// Zapisywanie trybu pracy HC1 do pamięci urządzenia
IF xTrybPracyHC1Zapisz AND (fbTaktowanieZapisywaniaModbus.Q OR rtrigZapisModbus.Q) THEN
	fnModbusZapisRejestru(	bAdresUrzadzenia := bAdres,
							bFunkcja := INT_TO_BYTE(enumModbusKodyFunkcji.ZapisRejestru),
							uiAdresRejestru := uintTrybPracyHC1AdresModbus,
							pZmiennaReferencyjna := 0,
							wWartoscDoZapisania := REAL_TO_WORD(rTrybPracyHC1Zapis),
							intModbusOdczytZapisZadanieRozmiar := intModbusOdczytZapisZadanieRozmiar,
							arModbusOdczytZapisZadanie := arModbusOdczytZapisZadanie,
							intModbusOdczytZapisZadanieZnacznikZapisu := intModbusOdczytZapisZadanieZnacznikZapisu);
	IF intTrybPracyHC1 = REAL_TO_INT(rTrybPracyHC1Zapis) THEN					
		xTrybPracyHC1Zapisz := FALSE;
	END_IF
END_IF
// Temperatura punktu X2 krzywej grzewczej HC1
IF xKrzywaGrzewczaTemperaturyZewnetrznejX2HC1Zapisz AND (fbTaktowanieZapisywaniaModbus.Q OR rtrigZapisModbus.Q) THEN
	wKrzywaGrzewczaTemperaturyZewnetrznejX2HC1Zapis := fnOdwrocenieBitowTemperaturyUjemnejREAL_TO_WORD(rTemperaturaKelviny := rKrzywaGrzewczaTemperaturyZewnetrznejX2HC1Zapis);
	fnModbusZapisRejestru(	bAdresUrzadzenia := bAdres,
							bFunkcja := INT_TO_BYTE(enumModbusKodyFunkcji.ZapisRejestru),
							uiAdresRejestru := uintKrzywaGrzewczaTemperaturyZewnetrznejX2HC1AdresModbus,
							pZmiennaReferencyjna := 0,
							wWartoscDoZapisania := wKrzywaGrzewczaTemperaturyZewnetrznejX2HC1Zapis,
							intModbusOdczytZapisZadanieRozmiar := intModbusOdczytZapisZadanieRozmiar,
							arModbusOdczytZapisZadanie := arModbusOdczytZapisZadanie,
							intModbusOdczytZapisZadanieZnacznikZapisu := intModbusOdczytZapisZadanieZnacznikZapisu);
	IF rKrzywaGrzewczaTemperaturyZewnetrznejX2HC1 = rKrzywaGrzewczaTemperaturyZewnetrznejX2HC1Zapis THEN 						
		xKrzywaGrzewczaTemperaturyZewnetrznejX2HC1Zapisz := FALSE;
	END_IF
END_IF
// Temperatura punktu X3 krzywej grzewczej HC1
IF xKrzywaGrzewczaTemperaturyZewnetrznejX3HC1Zapisz AND (fbTaktowanieZapisywaniaModbus.Q OR rtrigZapisModbus.Q) THEN
	wKrzywaGrzewczaTemperaturyZewnetrznejX3HC1Zapis := fnOdwrocenieBitowTemperaturyUjemnejREAL_TO_WORD(rTemperaturaKelviny := rKrzywaGrzewczaTemperaturyZewnetrznejX3HC1Zapis);
	fnModbusZapisRejestru(	bAdresUrzadzenia := bAdres,
							bFunkcja := INT_TO_BYTE(enumModbusKodyFunkcji.ZapisRejestru),
							uiAdresRejestru := uintKrzywaGrzewczaTemperaturyZewnetrznejX3HC1AdresModbus,
							pZmiennaReferencyjna := 0,
							wWartoscDoZapisania := wKrzywaGrzewczaTemperaturyZewnetrznejX3HC1Zapis,
							intModbusOdczytZapisZadanieRozmiar := intModbusOdczytZapisZadanieRozmiar,
							arModbusOdczytZapisZadanie := arModbusOdczytZapisZadanie,
							intModbusOdczytZapisZadanieZnacznikZapisu := intModbusOdczytZapisZadanieZnacznikZapisu);
	IF rKrzywaGrzewczaTemperaturyZewnetrznejX3HC1 = rKrzywaGrzewczaTemperaturyZewnetrznejX3HC1Zapis THEN 						
		xKrzywaGrzewczaTemperaturyZewnetrznejX3HC1Zapisz := FALSE;
	END_IF
END_IF
// Temperatura punktu X4 krzywej grzewczej HC1
IF xKrzywaGrzewczaTemperaturyZewnetrznejX4HC1Zapisz AND (fbTaktowanieZapisywaniaModbus.Q OR rtrigZapisModbus.Q) THEN
	wKrzywaGrzewczaTemperaturyZewnetrznejX4HC1Zapis := fnOdwrocenieBitowTemperaturyUjemnejREAL_TO_WORD(rTemperaturaKelviny := rKrzywaGrzewczaTemperaturyZewnetrznejX4HC1Zapis);
	fnModbusZapisRejestru(	bAdresUrzadzenia := bAdres,
							bFunkcja := INT_TO_BYTE(enumModbusKodyFunkcji.ZapisRejestru),
							uiAdresRejestru := uintKrzywaGrzewczaTemperaturyZewnetrznejX4HC1AdresModbus,
							pZmiennaReferencyjna := 0,
							wWartoscDoZapisania := wKrzywaGrzewczaTemperaturyZewnetrznejX4HC1Zapis,
							intModbusOdczytZapisZadanieRozmiar := intModbusOdczytZapisZadanieRozmiar,
							arModbusOdczytZapisZadanie := arModbusOdczytZapisZadanie,
							intModbusOdczytZapisZadanieZnacznikZapisu := intModbusOdczytZapisZadanieZnacznikZapisu);
	IF rKrzywaGrzewczaTemperaturyZewnetrznejX4HC1 = rKrzywaGrzewczaTemperaturyZewnetrznejX4HC1Zapis THEN 						
		xKrzywaGrzewczaTemperaturyZewnetrznejX4HC1Zapisz := FALSE;
	END_IF
END_IF
// Temperatura punktu X5 krzywej grzewczej HC1
IF xKrzywaGrzewczaTemperaturyZewnetrznejX5HC1Zapisz AND (fbTaktowanieZapisywaniaModbus.Q OR rtrigZapisModbus.Q) THEN
	wKrzywaGrzewczaTemperaturyZewnetrznejX5HC1Zapis := fnOdwrocenieBitowTemperaturyUjemnejREAL_TO_WORD(rTemperaturaKelviny := rKrzywaGrzewczaTemperaturyZewnetrznejX5HC1Zapis);
	fnModbusZapisRejestru(	bAdresUrzadzenia := bAdres,
							bFunkcja := INT_TO_BYTE(enumModbusKodyFunkcji.ZapisRejestru),
							uiAdresRejestru := uintKrzywaGrzewczaTemperaturyZewnetrznejX5HC1AdresModbus,
							pZmiennaReferencyjna := 0,
							wWartoscDoZapisania := wKrzywaGrzewczaTemperaturyZewnetrznejX5HC1Zapis,
							intModbusOdczytZapisZadanieRozmiar := intModbusOdczytZapisZadanieRozmiar,
							arModbusOdczytZapisZadanie := arModbusOdczytZapisZadanie,
							intModbusOdczytZapisZadanieZnacznikZapisu := intModbusOdczytZapisZadanieZnacznikZapisu);
	IF rKrzywaGrzewczaTemperaturyZewnetrznejX5HC1 = rKrzywaGrzewczaTemperaturyZewnetrznejX5HC1Zapis THEN 						
		xKrzywaGrzewczaTemperaturyZewnetrznejX5HC1Zapisz := FALSE;
	END_IF
END_IF
// Temperatura punktu X6 krzywej grzewczej HC1
IF xKrzywaGrzewczaTemperaturyZewnetrznejX6HC1Zapisz AND (fbTaktowanieZapisywaniaModbus.Q OR rtrigZapisModbus.Q) THEN
	wKrzywaGrzewczaTemperaturyZewnetrznejX6HC1Zapis := fnOdwrocenieBitowTemperaturyUjemnejREAL_TO_WORD(rTemperaturaKelviny := rKrzywaGrzewczaTemperaturyZewnetrznejX6HC1Zapis);
	fnModbusZapisRejestru(	bAdresUrzadzenia := bAdres,
							bFunkcja := INT_TO_BYTE(enumModbusKodyFunkcji.ZapisRejestru),
							uiAdresRejestru := uintKrzywaGrzewczaTemperaturyZewnetrznejX6HC1AdresModbus,
							pZmiennaReferencyjna := 0,
							wWartoscDoZapisania := wKrzywaGrzewczaTemperaturyZewnetrznejX6HC1Zapis,
							intModbusOdczytZapisZadanieRozmiar := intModbusOdczytZapisZadanieRozmiar,
							arModbusOdczytZapisZadanie := arModbusOdczytZapisZadanie,
							intModbusOdczytZapisZadanieZnacznikZapisu := intModbusOdczytZapisZadanieZnacznikZapisu);
	IF rKrzywaGrzewczaTemperaturyZewnetrznejX6HC1 = rKrzywaGrzewczaTemperaturyZewnetrznejX6HC1Zapis THEN 						
		xKrzywaGrzewczaTemperaturyZewnetrznejX6HC1Zapisz := FALSE;
	END_IF
END_IF
// Temperatura punktu Y2 krzywej grzewczej HC1
IF xKrzywaGrzewczaTemperaturyZasilaniaY2HC1Zapisz AND (fbTaktowanieZapisywaniaModbus.Q OR rtrigZapisModbus.Q) THEN
	fnModbusZapisRejestru(	bAdresUrzadzenia := bAdres,
							bFunkcja := INT_TO_BYTE(enumModbusKodyFunkcji.ZapisRejestru),
							uiAdresRejestru := uintKrzywaGrzewczaTemperaturyZasilaniaY2HC1AdresModbus,
							pZmiennaReferencyjna := 0,
							wWartoscDoZapisania := REAL_TO_WORD((rKrzywaGrzewczaTemperaturyZasilaniaY2HC1Zapis - 273.15) * 10),
							intModbusOdczytZapisZadanieRozmiar := intModbusOdczytZapisZadanieRozmiar,
							arModbusOdczytZapisZadanie := arModbusOdczytZapisZadanie,
							intModbusOdczytZapisZadanieZnacznikZapisu := intModbusOdczytZapisZadanieZnacznikZapisu);
	IF rKrzywaGrzewczaTemperaturyZasilaniaY2HC1 = rKrzywaGrzewczaTemperaturyZasilaniaY2HC1Zapis THEN 						
		xKrzywaGrzewczaTemperaturyZasilaniaY2HC1Zapisz := FALSE;
	END_IF
END_IF
// Temperatura punktu Y3 krzywej grzewczej HC1
IF xKrzywaGrzewczaTemperaturyZasilaniaY3HC1Zapisz AND (fbTaktowanieZapisywaniaModbus.Q OR rtrigZapisModbus.Q) THEN
	fnModbusZapisRejestru(	bAdresUrzadzenia := bAdres,
							bFunkcja := INT_TO_BYTE(enumModbusKodyFunkcji.ZapisRejestru),
							uiAdresRejestru := uintKrzywaGrzewczaTemperaturyZasilaniaY3HC1AdresModbus,
							pZmiennaReferencyjna := 0,
							wWartoscDoZapisania := REAL_TO_WORD((rKrzywaGrzewczaTemperaturyZasilaniaY3HC1Zapis - 273.15) * 10),
							intModbusOdczytZapisZadanieRozmiar := intModbusOdczytZapisZadanieRozmiar,
							arModbusOdczytZapisZadanie := arModbusOdczytZapisZadanie,
							intModbusOdczytZapisZadanieZnacznikZapisu := intModbusOdczytZapisZadanieZnacznikZapisu);
	IF rKrzywaGrzewczaTemperaturyZasilaniaY3HC1 = rKrzywaGrzewczaTemperaturyZasilaniaY3HC1Zapis THEN 						
		xKrzywaGrzewczaTemperaturyZasilaniaY3HC1Zapisz := FALSE;
	END_IF
END_IF
// Temperatura punktu Y4 krzywej grzewczej HC1
IF xKrzywaGrzewczaTemperaturyZasilaniaY4HC1Zapisz AND (fbTaktowanieZapisywaniaModbus.Q OR rtrigZapisModbus.Q) THEN
	fnModbusZapisRejestru(	bAdresUrzadzenia := bAdres,
							bFunkcja := INT_TO_BYTE(enumModbusKodyFunkcji.ZapisRejestru),
							uiAdresRejestru := uintKrzywaGrzewczaTemperaturyZasilaniaY4HC1AdresModbus,
							pZmiennaReferencyjna := 0,
							wWartoscDoZapisania := REAL_TO_WORD((rKrzywaGrzewczaTemperaturyZasilaniaY4HC1Zapis - 273.15) * 10),
							intModbusOdczytZapisZadanieRozmiar := intModbusOdczytZapisZadanieRozmiar,
							arModbusOdczytZapisZadanie := arModbusOdczytZapisZadanie,
							intModbusOdczytZapisZadanieZnacznikZapisu := intModbusOdczytZapisZadanieZnacznikZapisu);
	IF rKrzywaGrzewczaTemperaturyZasilaniaY4HC1 = rKrzywaGrzewczaTemperaturyZasilaniaY4HC1Zapis THEN 						
		xKrzywaGrzewczaTemperaturyZasilaniaY4HC1Zapisz := FALSE;
	END_IF
END_IF
// Temperatura punktu Y5 krzywej grzewczej HC1
IF xKrzywaGrzewczaTemperaturyZasilaniaY5HC1Zapisz AND (fbTaktowanieZapisywaniaModbus.Q OR rtrigZapisModbus.Q) THEN
	fnModbusZapisRejestru(	bAdresUrzadzenia := bAdres,
							bFunkcja := INT_TO_BYTE(enumModbusKodyFunkcji.ZapisRejestru),
							uiAdresRejestru := uintKrzywaGrzewczaTemperaturyZasilaniaY5HC1AdresModbus,
							pZmiennaReferencyjna := 0,
							wWartoscDoZapisania := REAL_TO_WORD((rKrzywaGrzewczaTemperaturyZasilaniaY5HC1Zapis - 273.15) * 10),
							intModbusOdczytZapisZadanieRozmiar := intModbusOdczytZapisZadanieRozmiar,
							arModbusOdczytZapisZadanie := arModbusOdczytZapisZadanie,
							intModbusOdczytZapisZadanieZnacznikZapisu := intModbusOdczytZapisZadanieZnacznikZapisu);
	IF rKrzywaGrzewczaTemperaturyZasilaniaY5HC1 = rKrzywaGrzewczaTemperaturyZasilaniaY5HC1Zapis THEN 						
		xKrzywaGrzewczaTemperaturyZasilaniaY5HC1Zapisz := FALSE;
	END_IF
END_IF
// Temperatura punktu Y6 krzywej grzewczej HC1
IF xKrzywaGrzewczaTemperaturyZasilaniaY6HC1Zapisz AND (fbTaktowanieZapisywaniaModbus.Q OR rtrigZapisModbus.Q) THEN
	fnModbusZapisRejestru(	bAdresUrzadzenia := bAdres,
							bFunkcja := INT_TO_BYTE(enumModbusKodyFunkcji.ZapisRejestru),
							uiAdresRejestru := uintKrzywaGrzewczaTemperaturyZasilaniaY6HC1AdresModbus,
							pZmiennaReferencyjna := 0,
							wWartoscDoZapisania := REAL_TO_WORD((rKrzywaGrzewczaTemperaturyZasilaniaY6HC1Zapis - 273.15) * 10),
							intModbusOdczytZapisZadanieRozmiar := intModbusOdczytZapisZadanieRozmiar,
							arModbusOdczytZapisZadanie := arModbusOdczytZapisZadanie,
							intModbusOdczytZapisZadanieZnacznikZapisu := intModbusOdczytZapisZadanieZnacznikZapisu);
	IF rKrzywaGrzewczaTemperaturyZasilaniaY6HC1 = rKrzywaGrzewczaTemperaturyZasilaniaY6HC1Zapis THEN 						
		xKrzywaGrzewczaTemperaturyZasilaniaY6HC1Zapisz := FALSE;
	END_IF				
END_IF
// Zapisywanie trybu pracy DHW do pamięci urządzenia
IF xTrybPracyDHWZapisz AND (fbTaktowanieZapisywaniaModbus.Q OR rtrigZapisModbus.Q) THEN
	fnModbusZapisRejestru(	bAdresUrzadzenia := bAdres,
							bFunkcja := INT_TO_BYTE(enumModbusKodyFunkcji.ZapisRejestru),
							uiAdresRejestru := uintTrybPracyZadanieDHWAdresModbus,
							pZmiennaReferencyjna := 0,
							wWartoscDoZapisania := REAL_TO_WORD(rTrybPracyDHWZapis),
							intModbusOdczytZapisZadanieRozmiar := intModbusOdczytZapisZadanieRozmiar,
							arModbusOdczytZapisZadanie := arModbusOdczytZapisZadanie,
							intModbusOdczytZapisZadanieZnacznikZapisu := intModbusOdczytZapisZadanieZnacznikZapisu);
	IF intTrybPracyDHW = REAL_TO_INT(rTrybPracyDHWZapis) THEN					
		xTrybPracyDHWZapisz := FALSE;
	END_IF
END_IF

// Wyznaczanie okresu grzewczego
fbZegar15M(IN := NOT fbZegar15M.Q AND NOT xBladBrakZmianyTemperaturyZewnetrznej, PT := T#15M);

	// Obliczenie wschodu i zachodu słońca
fbWschodZachod(dtUTC_Time := WagoAppTime.FuGetDateAndTime(),
	rTimeZone := 0,
	xDST := FALSE,
	rLatitude := 54.441944,
	rLongitude := 18.559722);

	// Zapisywanie tempratury z 15-minutowym okresem, oraz obliczanie średniej
IF fbWschodZachod.dtUTC_Time > fbWschodZachod.dtSunrise AND fbWschodZachod.dtUTC_Time < fbWschodZachod.dtSunset THEN
	IF fbZegar15M.Q OR xPierwszySkan THEN
		aTemperatury[iTemperaturyIndex] := WORD_TO_REAL(wTemperaturaZewnetrzna) / 10;
		iTemperaturyIndex := iTemperaturyIndex + 1;
	END_IF	
	xObliczSrednia3Dni := TRUE;
ELSE 
	// Obliczanie średniej temperatury dziennej
	IF iTemperaturyIndex >= 40 THEN		// Oblicz średnią temperaturę tylko, jeśli zebranych zostało przynajmniej 40 próbek
		rTemperaturaSrednia1Dzien := 0;
		iIloscPomiarow := iTemperaturyIndex;
		FOR iTemperaturyIndex := 0 TO iIloscPomiarow BY 1 DO  
			rTemperaturaSrednia1Dzien := rTemperaturaSrednia1Dzien + aTemperatury[iTemperaturyIndex];
		END_FOR
		rTemperaturaSrednia1Dzien := rTemperaturaSrednia1Dzien / iTemperaturyIndex;
		xBladIloscPomiarowTemperatury := FALSE;
	ELSE
		rTemperaturaSrednia1Dzien := 15;
		xBladIloscPomiarowTemperatury := TRUE;
	END_IF
	// Obliczanie średniej z trzech dni
	IF xObliczSrednia3Dni THEN
		aTemperaturySrednie[iTemperaturySrednieIndex] := rTemperaturaSrednia1Dzien;
		iTemperaturySrednieIndex := iTemperaturySrednieIndex + 1;
		IF iTemperaturySrednieIndex = 3 THEN 
			iTemperaturySrednieIndex := 0;
			xTemperaturaSrednia3DniObliczona := TRUE;
		END_IF
		rTemperaturaSrednia3Dni := (aTemperaturySrednie[0] + aTemperaturySrednie[1] + aTemperaturySrednie[2]) / 3; 
		xObliczSrednia3Dni := FALSE;	
	END_IF
	iTemperaturyIndex := 0;
END_IF

	// Sprawdzenie warunku na włączenie ogrzewania (pomiędzy 15 września a 15 maja i/lub średnia temperatura jest poniżej 15 stopni)
IF  ((fbWschodZachod._rDay >= 15 AND fbWschodZachod._rMonth = 9) OR (fbWschodZachod._rMonth > 9 OR fbWschodZachod._rMonth < 5) OR (fbWschodZachod._rDay <= 15 AND fbWschodZachod._rMonth = 5)) OR 
	(rTemperaturaSrednia3Dni < 15 AND xTemperaturaSrednia3DniObliczona) OR xSezonGrzewczyCalyRok THEN
	xSezonGrzewczy := TRUE;
	intTrybPracyHC1Autonomizacja := enumPPPSWezelClimatixPOL63xTrybPracy.Komfort;
ELSE
	xSezonGrzewczy := FALSE;
	intTrybPracyHC1Autonomizacja := enumPPPSWezelClimatixPOL63xTrybPracy.OchronaBudynku;
END_IF

// dokonywanie obliczeń
(*
xOdczytanaKlasaAlarmuBezpieczenstwa := WORD_TO_BOOL(wOdczytanaKlasaAlarmuBezpieczenstwa);
xOdczytanaKlasaAlarmuKrytyczny := WORD_TO_BOOL(wOdczytanaKlasaAlarmuKrytyczny);
xOdczytanaKlasaAlarmuOstrzezenie := WORD_TO_BOOL(wOdczytanaKlasaAlarmuOstrzezenie);
xOdczytanaKlasaAlarmuInformacyjny := WORD_TO_BOOL(wOdczytanaKlasaAlarmuInformacyjny);
*)
xReczneWylaczenieInstalacji := WORD_TO_BOOL(wReczneWylaczenieInstalacji);

IF xInstalacjaHC1 OR xInstalacjaHC2 THEN
	fbTemperaturaZewnetrzna(	rWartoscWejsciowa := WORD_TO_REAL(wTemperaturaZewnetrzna),
									rDeadband := 0.5,
									tCzasMinimalny := tMinimalnyCzasRaportowania,
									tCzasMaksymalny := tMaksymalnyCzasRaportowania,
									rWynikMnoznik := 0.1,
									rWynikOffset := 273.15,
									rWartoscWejsciowaZaraportowana := rTemperaturaZewnetrznaZaraportowana,
									rWartoscWyjsciowa => rTemperaturaZewnetrzna);
END_IF

IF xInstalacjaHC1 THEN							
	fbTemperaturaGrzaniaNastawionaHC1(	rWartoscWejsciowa := WORD_TO_REAL(wTemperaturaGrzaniaNastawionaHC1),
									rDeadband := 0.5,
									tCzasMinimalny := tMinimalnyCzasRaportowania,
									tCzasMaksymalny := tMaksymalnyCzasRaportowania,
									rWynikMnoznik := 0.1,
									rWynikOffset := 273.15,
									rWartoscWejsciowaZaraportowana := rTemperaturaGrzaniaNastawionaHC1Zaraportowana,
									rWartoscWyjsciowa => rTemperaturaGrzaniaNastawionaHC1);
						
	fbTemperaturaGrzaniaNastawionaKrzywaGrzewczaHC1(	rWartoscWejsciowa := WORD_TO_REAL(wTemperaturaGrzaniaNastawionaKrzywaGrzewczaHC1),
									rDeadband := 0.5,
									tCzasMinimalny := tMinimalnyCzasRaportowania,
									tCzasMaksymalny := tMaksymalnyCzasRaportowania,
									rWynikMnoznik := 0.1,
									rWynikOffset := 273.15,
									rWartoscWejsciowaZaraportowana := rTemperaturaGrzaniaNastawionaKrzywaGrzewczaHC1Zaraportowana,
									rWartoscWyjsciowa => rTemperaturaGrzaniaNastawionaHC1);
	
	IF xReczneWylaczenieInstalacji THEN
		intTrybPracyHC1 := enumPPPSWezelClimatixPOL63xTrybPracy.ReczneWylaczenie;
	ELSE
		IF wTrybPracyHC1 = 0 THEN
			intTrybPracyHC1 := enumPPPSWezelClimatixPOL63xTrybPracy.Auto;
		ELSE
			IF wTrybPracyHC1 = 1 THEN
				intTrybPracyHC1 := enumPPPSWezelClimatixPOL63xTrybPracy.OchronaBudynku;
			ELSE
				IF wTrybPracyHC1 = 2 THEN
					intTrybPracyHC1 := enumPPPSWezelClimatixPOL63xTrybPracy.Ekonomiczny;
				ELSE
					IF wTrybPracyHC1 = 3 THEN
						intTrybPracyHC1 := enumPPPSWezelClimatixPOL63xTrybPracy.Komfort;
					END_IF
				END_IF
			END_IF
		END_IF
	END_IF
					
	fbTemperaturaGrzaniaNastawionaHC1(	rWartoscWejsciowa := WORD_TO_REAL(wTemperaturaGrzaniaNastawionaHC1),
									rDeadband := 0.5,
									tCzasMinimalny := tMinimalnyCzasRaportowania,
									tCzasMaksymalny := tMaksymalnyCzasRaportowania,
									rWynikMnoznik := 0.1,
									rWynikOffset := 273.15,
									rWartoscWejsciowaZaraportowana := rTemperaturaGrzaniaNastawionaHC1Zaraportowana,
									rWartoscWyjsciowa => rTemperaturaGrzaniaNastawionaHC1);

	fbTemperaturaGrzaniaNastawionaKrzywaGrzewczaHC1(	rWartoscWejsciowa := WORD_TO_REAL(wTemperaturaGrzaniaNastawionaKrzywaGrzewczaHC1),
									rDeadband := 0.5,
									tCzasMinimalny := tMinimalnyCzasRaportowania,
									tCzasMaksymalny := tMaksymalnyCzasRaportowania,
									rWynikMnoznik := 0.1,
									rWynikOffset := 273.15,
									rWartoscWejsciowaZaraportowana := rTemperaturaGrzaniaNastawionaKrzywaGrzewczaHC1Zaraportowana,
									rWartoscWyjsciowa => rTemperaturaGrzaniaNastawionaKrzywaGrzewczaHC1);
								
	fbTemperaturaZasilaniaObwoduHC1(	rWartoscWejsciowa := WORD_TO_REAL(wTemperaturaZasilaniaObwoduHC1),
									rDeadband := 0.5,
									tCzasMinimalny := tMinimalnyCzasRaportowania,
									tCzasMaksymalny := tMaksymalnyCzasRaportowania,
									rWynikMnoznik := 0.1,
									rWynikOffset := 273.15,
									rWartoscWejsciowaZaraportowana := rTemperaturaZasilaniaObwoduHC1Zaraportowana,
									rWartoscWyjsciowa => rTemperaturaZasilaniaObwoduHC1);
									
	fbTemperaturaPowrotuObwoduHC1(	rWartoscWejsciowa := WORD_TO_REAL(wTemperaturaPowrotuObwoduHC1),
									rDeadband := 0.5,
									tCzasMinimalny := tMinimalnyCzasRaportowania,
									tCzasMaksymalny := tMaksymalnyCzasRaportowania,
									rWynikMnoznik := 0.1,
									rWynikOffset := 273.15,
									rWartoscWejsciowaZaraportowana := rTemperaturaPowrotuObwoduHC1Zaraportowana,
									rWartoscWyjsciowa => rTemperaturaPowrotuObwoduHC1);
									
	fbTemperaturaPowrotuMiastoHC1(	rWartoscWejsciowa := WORD_TO_REAL(wTemperaturaPowrotuMiastoHC1),
									rDeadband := 0.5,
									tCzasMinimalny := tMinimalnyCzasRaportowania,
									tCzasMaksymalny := tMaksymalnyCzasRaportowania,
									rWynikMnoznik := 0.1,
									rWynikOffset := 273.15,
									rWartoscWejsciowaZaraportowana := rTemperaturaPowrotuMiastoHC1Zaraportowana,
									rWartoscWyjsciowa => rTemperaturaPowrotuMiastoHC1);
									
	fbTemperaturaZasilaniaBudynku(	rWartoscWejsciowa := WORD_TO_REAL(wTemperaturaZasilaniaBudynku),
									rDeadband := 0.5,
									tCzasMinimalny := tMinimalnyCzasRaportowania,
									tCzasMaksymalny := tMaksymalnyCzasRaportowania,
									rWynikMnoznik := 0.1,
									rWynikOffset := 273.15,
									rWartoscWejsciowaZaraportowana := rTemperaturaZasilaniaBudynkuZaraportowana,
									rWartoscWyjsciowa => rTemperaturaZasilaniaBudynku);
									
	fbTemperaturaPowrotuBudynku(	rWartoscWejsciowa := WORD_TO_REAL(wTemperaturaPowrotuBudynku),
									rDeadband := 0.5,
									tCzasMinimalny := tMinimalnyCzasRaportowania,
									tCzasMaksymalny := tMaksymalnyCzasRaportowania,
									rWynikMnoznik := 0.1,
									rWynikOffset := 273.15,
									rWartoscWejsciowaZaraportowana := rTemperaturaPowrotuBudynkuZaraportowana,
									rWartoscWyjsciowa => rTemperaturaPowrotuBudynku);
									
	fbSygnalZadaniaGrzaniaHC1(	rWartoscWejsciowa := WORD_TO_REAL(wSygnalZadaniaGrzaniaHC1),
									rDeadband := 0.05,
									tCzasMinimalny := tMinimalnyCzasRaportowania,
									tCzasMaksymalny := tMaksymalnyCzasRaportowania,
									rWynikMnoznik := 0.01,
									rWynikOffset := 0.0,
									rWartoscWejsciowaZaraportowana := rSygnalZadaniaGrzaniaHC1Zaraportowana,
									rWartoscWyjsciowa => rSygnalZadaniaGrzaniaHC1);
									
	fbStopienOtwarciaZaworuMiastoHC1(	rWartoscWejsciowa := WORD_TO_REAL(wStopienOtwarciaZaworuMiastoHC1),
									rDeadband := 0.05,
									tCzasMinimalny := tMinimalnyCzasRaportowania,
									tCzasMaksymalny := tMaksymalnyCzasRaportowania,
									rWynikMnoznik := 0.01,
									rWynikOffset := 0.0,
									rWartoscWejsciowaZaraportowana := rStopienOtwarciaZaworuMiastoHC1Zaraportowana,
									rWartoscWyjsciowa => rStopienOtwarciaZaworuMiastoHC1);
									
	IF wKrzywaGrzewczaTemperaturyZewnetrznejX2OdczytHC1 > 1000 THEN		// Jeśli temperatura ujemna odwróć bity	
		rKrzywaGrzewczaTemperaturyZewnetrznejX2HC1Raport := (-1) * WORD_TO_REAL(wKrzywaGrzewczaTemperaturyZewnetrznejX2OdczytHC1 XOR 16#FFFF);	
	ELSE
		rKrzywaGrzewczaTemperaturyZewnetrznejX2HC1Raport := WORD_TO_REAL(wKrzywaGrzewczaTemperaturyZewnetrznejX2OdczytHC1);
	END_IF		
	fbKrzywaGrzewczaTemperaturyZewnetrznejX2HC1(	rWartoscWejsciowa := rKrzywaGrzewczaTemperaturyZewnetrznejX2HC1Raport,
									rDeadband := 0.5,
									tCzasMinimalny := tMinimalnyCzasRaportowania,
									tCzasMaksymalny := tMaksymalnyCzasRaportowania,
									rWynikMnoznik := 0.1,
									rWynikOffset := 273.15,
									rWartoscWejsciowaZaraportowana := rKrzywaGrzewczaTemperaturyZewnetrznejX2HC1Zaraportowana,
									rWartoscWyjsciowa => rKrzywaGrzewczaTemperaturyZewnetrznejX2HC1);
	
	fbKrzywaGrzewczaTemperaturyZasilaniaY2HC1(	rWartoscWejsciowa := WORD_TO_REAL(wKrzywaGrzewczaTemperaturyZasilaniaY2OdczytHC1),
									rDeadband := 0.5,
									tCzasMinimalny := tMinimalnyCzasRaportowania,
									tCzasMaksymalny := tMaksymalnyCzasRaportowania,
									rWynikMnoznik := 0.1,
									rWynikOffset := 273.15,
									rWartoscWejsciowaZaraportowana := rKrzywaGrzewczaTemperaturyZasilaniaY2HC1Zaraportowana,
									rWartoscWyjsciowa => rKrzywaGrzewczaTemperaturyZasilaniaY2HC1);
	
	IF wKrzywaGrzewczaTemperaturyZewnetrznejX3OdczytHC1 > 1000 THEN		// Jeśli temperatura ujemna odwróć bity	
		rKrzywaGrzewczaTemperaturyZewnetrznejX3HC1Raport := (-1) * WORD_TO_REAL(wKrzywaGrzewczaTemperaturyZewnetrznejX3OdczytHC1 XOR 16#FFFF);	
	ELSE
		rKrzywaGrzewczaTemperaturyZewnetrznejX3HC1Raport := WORD_TO_REAL(wKrzywaGrzewczaTemperaturyZewnetrznejX3OdczytHC1);
	END_IF								
	fbKrzywaGrzewczaTemperaturyZewnetrznejX3HC1(	rWartoscWejsciowa := rKrzywaGrzewczaTemperaturyZewnetrznejX3HC1Raport,
									rDeadband := 0.5,
									tCzasMinimalny := tMinimalnyCzasRaportowania,
									tCzasMaksymalny := tMaksymalnyCzasRaportowania,
									rWynikMnoznik := 0.1,
									rWynikOffset := 273.15,
									rWartoscWejsciowaZaraportowana := rKrzywaGrzewczaTemperaturyZewnetrznejX3HC1Zaraportowana,
									rWartoscWyjsciowa => rKrzywaGrzewczaTemperaturyZewnetrznejX3HC1);
	
	fbKrzywaGrzewczaTemperaturyZasilaniaY3HC1(	rWartoscWejsciowa := WORD_TO_REAL(wKrzywaGrzewczaTemperaturyZasilaniaY3OdczytHC1),
									rDeadband := 0.5,
									tCzasMinimalny := tMinimalnyCzasRaportowania,
									tCzasMaksymalny := tMaksymalnyCzasRaportowania,
									rWynikMnoznik := 0.1,
									rWynikOffset := 273.15,
									rWartoscWejsciowaZaraportowana := rKrzywaGrzewczaTemperaturyZasilaniaY3HC1Zaraportowana,
									rWartoscWyjsciowa => rKrzywaGrzewczaTemperaturyZasilaniaY3HC1);
	
	IF wKrzywaGrzewczaTemperaturyZewnetrznejX4OdczytHC1 > 1000 THEN		// Jeśli temperatura ujemna odwróć bity	
		rKrzywaGrzewczaTemperaturyZewnetrznejX4HC1Raport := (-1) * WORD_TO_REAL(wKrzywaGrzewczaTemperaturyZewnetrznejX4OdczytHC1 XOR 16#FFFF);	
	ELSE
		rKrzywaGrzewczaTemperaturyZewnetrznejX4HC1Raport := WORD_TO_REAL(wKrzywaGrzewczaTemperaturyZewnetrznejX4OdczytHC1);
	END_IF												
	fbKrzywaGrzewczaTemperaturyZewnetrznejX4HC1(	rWartoscWejsciowa := rKrzywaGrzewczaTemperaturyZewnetrznejX4HC1Raport,
									rDeadband := 0.5,
									tCzasMinimalny := tMinimalnyCzasRaportowania,
									tCzasMaksymalny := tMaksymalnyCzasRaportowania,
									rWynikMnoznik := 0.1,
									rWynikOffset := 273.15,
									rWartoscWejsciowaZaraportowana := rKrzywaGrzewczaTemperaturyZewnetrznejX4HC1Zaraportowana,
									rWartoscWyjsciowa => rKrzywaGrzewczaTemperaturyZewnetrznejX4HC1);
	
	fbKrzywaGrzewczaTemperaturyZasilaniaY4HC1(	rWartoscWejsciowa := WORD_TO_REAL(wKrzywaGrzewczaTemperaturyZasilaniaY4OdczytHC1),
									rDeadband := 0.5,
									tCzasMinimalny := tMinimalnyCzasRaportowania,
									tCzasMaksymalny := tMaksymalnyCzasRaportowania,
									rWynikMnoznik := 0.1,
									rWynikOffset := 273.15,
									rWartoscWejsciowaZaraportowana := rKrzywaGrzewczaTemperaturyZasilaniaY4HC1Zaraportowana,
									rWartoscWyjsciowa => rKrzywaGrzewczaTemperaturyZasilaniaY4HC1);
	
		
	IF wKrzywaGrzewczaTemperaturyZewnetrznejX5OdczytHC1 > 1000 THEN		// Jeśli temperatura ujemna odwróć bity	
		rKrzywaGrzewczaTemperaturyZewnetrznejX5HC1Raport := (-1) * WORD_TO_REAL(wKrzywaGrzewczaTemperaturyZewnetrznejX5OdczytHC1 XOR 16#FFFF);	
	ELSE
		rKrzywaGrzewczaTemperaturyZewnetrznejX5HC1Raport := WORD_TO_REAL(wKrzywaGrzewczaTemperaturyZewnetrznejX5OdczytHC1);
	END_IF										
	fbKrzywaGrzewczaTemperaturyZewnetrznejX5HC1(	rWartoscWejsciowa := rKrzywaGrzewczaTemperaturyZewnetrznejX5HC1Raport,
									rDeadband := 0.5,
									tCzasMinimalny := tMinimalnyCzasRaportowania,
									tCzasMaksymalny := tMaksymalnyCzasRaportowania,
									rWynikMnoznik := 0.1,
									rWynikOffset := 273.15,
									rWartoscWejsciowaZaraportowana := rKrzywaGrzewczaTemperaturyZewnetrznejX5HC1Zaraportowana,
									rWartoscWyjsciowa => rKrzywaGrzewczaTemperaturyZewnetrznejX5HC1);
	
	fbKrzywaGrzewczaTemperaturyZasilaniaY5HC1(	rWartoscWejsciowa := WORD_TO_REAL(wKrzywaGrzewczaTemperaturyZasilaniaY5OdczytHC1),
									rDeadband := 0.5,
									tCzasMinimalny := tMinimalnyCzasRaportowania,
									tCzasMaksymalny := tMaksymalnyCzasRaportowania,
									rWynikMnoznik := 0.1,
									rWynikOffset := 273.15,
									rWartoscWejsciowaZaraportowana := rKrzywaGrzewczaTemperaturyZasilaniaY5HC1Zaraportowana,
									rWartoscWyjsciowa => rKrzywaGrzewczaTemperaturyZasilaniaY5HC1);
	
	IF wKrzywaGrzewczaTemperaturyZewnetrznejX6OdczytHC1 > 1000 THEN		// Jeśli temperatura ujemna odwróć bity	
		rKrzywaGrzewczaTemperaturyZewnetrznejX6HC1Raport := (-1) * WORD_TO_REAL(wKrzywaGrzewczaTemperaturyZewnetrznejX6OdczytHC1 XOR 16#FFFF);	
	ELSE
		rKrzywaGrzewczaTemperaturyZewnetrznejX6HC1Raport := WORD_TO_REAL(wKrzywaGrzewczaTemperaturyZewnetrznejX6OdczytHC1);
	END_IF									
	fbKrzywaGrzewczaTemperaturyZewnetrznejX6HC1(	rWartoscWejsciowa := rKrzywaGrzewczaTemperaturyZewnetrznejX6HC1Raport,
									rDeadband := 0.5,
									tCzasMinimalny := tMinimalnyCzasRaportowania,
									tCzasMaksymalny := tMaksymalnyCzasRaportowania,
									rWynikMnoznik := 0.1,
									rWynikOffset := 273.15,
									rWartoscWejsciowaZaraportowana := rKrzywaGrzewczaTemperaturyZewnetrznejX6HC1Zaraportowana,
									rWartoscWyjsciowa => rKrzywaGrzewczaTemperaturyZewnetrznejX6HC1);
	
	fbKrzywaGrzewczaTemperaturyZasilaniaY6HC1(	rWartoscWejsciowa := WORD_TO_REAL(wKrzywaGrzewczaTemperaturyZasilaniaY6OdczytHC1),
									rDeadband := 0.5,
									tCzasMinimalny := tMinimalnyCzasRaportowania,
									tCzasMaksymalny := tMaksymalnyCzasRaportowania,
									rWynikMnoznik := 0.1,
									rWynikOffset := 273.15,
									rWartoscWejsciowaZaraportowana := rKrzywaGrzewczaTemperaturyZasilaniaY6HC1Zaraportowana,
									rWartoscWyjsciowa => rKrzywaGrzewczaTemperaturyZasilaniaY6HC1);


	intTrybOperacjiHC1 := WORD_TO_INT(wTrybOperacjiHC1);
END_IF

IF xInstalacjaDHW THEN
	fbTemperaturaGrzaniaNastawionaDHW(	rWartoscWejsciowa := WORD_TO_REAL(wTemperaturaGrzaniaNastawionaDHW),
									rDeadband := 0.5,
									tCzasMinimalny := tMinimalnyCzasRaportowania,
									tCzasMaksymalny := tMaksymalnyCzasRaportowania,
									rWynikMnoznik := 0.1,
									rWynikOffset := 273.15,
									rWartoscWejsciowaZaraportowana := rTemperaturaGrzaniaNastawionaDHWZaraportowana,
									rWartoscWyjsciowa => rTemperaturaGrzaniaNastawionaDHW);
									
	IF xReczneWylaczenieInstalacji THEN
		intTrybPracyDHW := enumPPPSWezelClimatixPOL63xTrybPracy.ReczneWylaczenie;
	ELSE
		IF wTrybPracyDHW = 0 THEN
			intTrybPracyDHW := enumPPPSWezelClimatixPOL63xTrybPracy.Auto;
		ELSE
			IF wTrybPracyDHW = 1 THEN
				intTrybPracyDHW := enumPPPSWezelClimatixPOL63xTrybPracy.OchronaBudynku;
			ELSE
				IF wTrybPracyDHW = 2 THEN
					intTrybPracyDHW := enumPPPSWezelClimatixPOL63xTrybPracy.Ekonomiczny;
				ELSE
					IF wTrybPracyDHW = 3 THEN
						intTrybPracyDHW := enumPPPSWezelClimatixPOL63xTrybPracy.Komfort;
					END_IF
				END_IF
			END_IF
		END_IF
	END_IF
					
	fbTemperaturaPowrotuMiastoDHW(	rWartoscWejsciowa := WORD_TO_REAL(wTemperaturaPowrotuMiastoDHW),
									rDeadband := 0.5,
									tCzasMinimalny := tMinimalnyCzasRaportowania,
									tCzasMaksymalny := tMaksymalnyCzasRaportowania,
									rWynikMnoznik := 0.1,
									rWynikOffset := 273.15,
									rWartoscWejsciowaZaraportowana := rTemperaturaPowrotuMiastoDHWZaraportowana,
									rWartoscWyjsciowa => rTemperaturaPowrotuMiastoDHW);
									
	fbTemperaturaZasilaniaBudynekDHW(	rWartoscWejsciowa := WORD_TO_REAL(wTemperaturaZasilaniaBudynekDHW),
									rDeadband := 0.5,
									tCzasMinimalny := tMinimalnyCzasRaportowania,
									tCzasMaksymalny := tMaksymalnyCzasRaportowania,
									rWynikMnoznik := 0.1,
									rWynikOffset := 273.15,
									rWartoscWejsciowaZaraportowana := rTemperaturaZasilaniaBudynekDHWZaraportowana,
									rWartoscWyjsciowa => rTemperaturaZasilaniaBudynekDHW);
									
	fbTemperaturaPowrotuBudynekDHW(	rWartoscWejsciowa := WORD_TO_REAL(wTemperaturaPowrotuBudynekDHW),
									rDeadband := 0.5,
									tCzasMinimalny := tMinimalnyCzasRaportowania,
									tCzasMaksymalny := tMaksymalnyCzasRaportowania,
									rWynikMnoznik := 0.1,
									rWynikOffset := 273.15,
									rWartoscWejsciowaZaraportowana := rTemperaturaPowrotuBudynekDHWZaraportowana,
									rWartoscWyjsciowa => rTemperaturaPowrotuBudynekDHW);
									
	fbStopienOtwarciaZaworuMiastoDHW(	rWartoscWejsciowa := WORD_TO_REAL(wStopienOtwarciaZaworuMiastoDHW),
									rDeadband := 0.05,
									tCzasMinimalny := tMinimalnyCzasRaportowania,
									tCzasMaksymalny := tMaksymalnyCzasRaportowania,
									rWynikMnoznik := 0.01,
									rWynikOffset := 0.0,
									rWartoscWejsciowaZaraportowana := rStopienOtwarciaZaworuMiastoDHWZaraportowana,
									rWartoscWyjsciowa => rStopienOtwarciaZaworuMiastoDHW);
									
	intTrybOperacjiDHW := WORD_TO_INT(wTrybOperacjiDHW);
END_IF


//raportowanie
IF (intBlokadaWykonywaniaRozkazow <> intBlokadaWykonywaniaRozkazowZaraportowana OR rTemperaturaZewnetrzna <> rTemperaturaZewnetrznaZaraportowana OR rTemperaturaGrzaniaNastawionaHC1 <> rTemperaturaGrzaniaNastawionaHC1Zaraportowana
OR intTrybPracyHC1 <> intTrybPracyHC1Zaraportowana OR rTemperaturaZasilaniaObwoduHC1 <> rTemperaturaZasilaniaObwoduHC1Zaraportowana OR rTemperaturaPowrotuObwoduHC1 <> rTemperaturaPowrotuObwoduHC1Zaraportowana
OR rTemperaturaPowrotuMiastoHC1 <> rTemperaturaPowrotuMiastoHC1Zaraportowana OR rTemperaturaZasilaniaBudynku <> rTemperaturaZasilaniaBudynkuZaraportowana OR rTemperaturaPowrotuBudynku <> rTemperaturaPowrotuBudynkuZaraportowana
OR rSygnalZadaniaGrzaniaHC1 <> rSygnalZadaniaGrzaniaHC1Zaraportowana OR rStopienOtwarciaZaworuMiastoHC1 <> rStopienOtwarciaZaworuMiastoHC1Zaraportowana OR rKrzywaGrzewczaTemperaturyZewnetrznejX2HC1 <> rKrzywaGrzewczaTemperaturyZewnetrznejX2HC1Zaraportowana
OR rKrzywaGrzewczaTemperaturyZewnetrznejX2HC1 <> rKrzywaGrzewczaTemperaturyZewnetrznejX2HC1Zaraportowana OR rKrzywaGrzewczaTemperaturyZewnetrznejX3HC1 <> rKrzywaGrzewczaTemperaturyZewnetrznejX3HC1Zaraportowana OR rKrzywaGrzewczaTemperaturyZewnetrznejX4HC1 <> rKrzywaGrzewczaTemperaturyZewnetrznejX4HC1Zaraportowana
OR rKrzywaGrzewczaTemperaturyZewnetrznejX5HC1 <> rKrzywaGrzewczaTemperaturyZewnetrznejX5HC1Zaraportowana OR rKrzywaGrzewczaTemperaturyZewnetrznejX6HC1 <> rKrzywaGrzewczaTemperaturyZewnetrznejX6HC1Zaraportowana
OR rKrzywaGrzewczaTemperaturyZasilaniaY2HC1 <> rKrzywaGrzewczaTemperaturyZasilaniaY2HC1Zaraportowana OR rKrzywaGrzewczaTemperaturyZasilaniaY3HC1 <> rKrzywaGrzewczaTemperaturyZasilaniaY3HC1Zaraportowana OR rKrzywaGrzewczaTemperaturyZasilaniaY4HC1 <> rKrzywaGrzewczaTemperaturyZasilaniaY4HC1Zaraportowana
OR rKrzywaGrzewczaTemperaturyZasilaniaY5HC1 <> rKrzywaGrzewczaTemperaturyZasilaniaY5HC1Zaraportowana OR rKrzywaGrzewczaTemperaturyZasilaniaY6HC1 <> rKrzywaGrzewczaTemperaturyZasilaniaY6HC1Zaraportowana
OR rTemperaturaGrzaniaNastawionaDHW <> rTemperaturaGrzaniaNastawionaDHWZaraportowana OR intTrybPracyDHW <> intTrybPracyDHWZaraportowana OR rTemperaturaPowrotuMiastoDHW <> rTemperaturaPowrotuMiastoDHWZaraportowana
OR rTemperaturaZasilaniaBudynekDHW <> rTemperaturaZasilaniaBudynekDHWZaraportowana OR rTemperaturaPowrotuBudynekDHW <> rTemperaturaPowrotuBudynekDHWZaraportowana OR rStopienOtwarciaZaworuMiastoDHW <> rStopienOtwarciaZaworuMiastoDHWZaraportowana 
OR intTrybOperacjiHC1 <> intTrybOperacjiHC1Zaraportowana OR rTemperaturaGrzaniaNastawionaKrzywaGrzewczaHC1 <> rTemperaturaGrzaniaNastawionaKrzywaGrzewczaHC1Zaraportowana OR intTrybOperacjiDHW <> intTrybOperacjiDHWZaraportowana
OR intTrybOperacjiDHW <> intTrybOperacjiDHWZaraportowana OR wAlarmsWord1 <> wAlarmsWord1Zaraportowana OR wAlarmsWord2 <> wAlarmsWord2Zaraportowana OR wAlarmsWord3 <> wAlarmsWord3Zaraportowana
OR wAlarmsWord4 <> wAlarmsWord4Zaraportowana OR xSezonGrzewczy <> xSezonGrzewczyZaraportowana OR rTemperaturaSrednia1Dzien <> rTemperaturaSrednia1DzienZaraportowana) 
AND	arModbusStatusKomunikacji[bAdres] = enumModbusStatus.KomunikacjaPrawidlowa AND xPoInicjalizacji THEN
	xRaport := TRUE;
END_IF

IF xRaport THEN
	sDane := '';
	xRaport := FALSE;
	IF intBlokadaWykonywaniaRozkazow <> intBlokadaWykonywaniaRozkazowZaraportowana THEN
		intBlokadaWykonywaniaRozkazowZaraportowana := intBlokadaWykonywaniaRozkazow;
		fnKomunikatDaneDodaj_xOverFlow(sDane := sDane , sAtrybut := 'BLOK=' , sWartosc := INT_TO_STRING(intBlokadaWykonywaniaRozkazow) , xOverFlow := xOverFlow);	
			IF xOverFlow = TRUE THEN
				fnZapiszKomunikat(	sCalyKomunikat := '' ,
							sTypKomunikatu := 'A' ,
							sMnemonik := sMnemonik ,
							sMACAdres := sMACAdres ,
							sIDNadawcy := sIdInstancji ,
							sIDOdbiorcy := sIdAplikacji ,
							sDaneZapasowe := sDaneZapasowe ,
							sDane := sDane ,
							arTablicaKomunikatow := arTablicaKomunikatow ,
							intTablicaKomunikatowZnacznikZapisu := intTablicaKomunikatowZnacznikZapisu ,
							intTablicaKomunikatowRozmiar := intTablicaKomunikatowRozmiar ,
							sWyslanyKomunikat := sWyslanyKomunikatDummy);
				sDane := '';
			END_IF	
	END_IF	
	IF wAlarmsWord1 <> wAlarmsWord1Zaraportowana THEN
	wAlarmsWord1Zaraportowana := wAlarmsWord1;
	fnKomunikatDaneDodaj_xOverFlow(sDane := sDane , sAtrybut := 'ALARMWORD1=' , sWartosc := WORD_TO_STRING(wAlarmsWord1) , xOverFlow := xOverFlow);	
		IF xOverFlow = TRUE THEN
			fnZapiszKomunikat(	sCalyKomunikat := '' ,
						sTypKomunikatu := 'A' ,
						sMnemonik := sMnemonik ,
						sMACAdres := sMACAdres ,
						sIDNadawcy := sIdInstancji ,
						sIDOdbiorcy := sIdAplikacji ,
						sDaneZapasowe := sDaneZapasowe ,
						sDane := sDane ,
						arTablicaKomunikatow := arTablicaKomunikatow ,
						intTablicaKomunikatowZnacznikZapisu := intTablicaKomunikatowZnacznikZapisu ,
						intTablicaKomunikatowRozmiar := intTablicaKomunikatowRozmiar ,
						sWyslanyKomunikat := sWyslanyKomunikatDummy);
			sDane := '';
		END_IF	
	END_IF	
	IF wAlarmsWord2 <> wAlarmsWord2Zaraportowana THEN
	wAlarmsWord2Zaraportowana := wAlarmsWord2;
	fnKomunikatDaneDodaj_xOverFlow(sDane := sDane , sAtrybut := 'ALARMWORD2=' , sWartosc := WORD_TO_STRING(wAlarmsWord2) , xOverFlow := xOverFlow);	
		IF xOverFlow = TRUE THEN
			fnZapiszKomunikat(	sCalyKomunikat := '' ,
						sTypKomunikatu := 'A' ,
						sMnemonik := sMnemonik ,
						sMACAdres := sMACAdres ,
						sIDNadawcy := sIdInstancji ,
						sIDOdbiorcy := sIdAplikacji ,
						sDaneZapasowe := sDaneZapasowe ,
						sDane := sDane ,
						arTablicaKomunikatow := arTablicaKomunikatow ,
						intTablicaKomunikatowZnacznikZapisu := intTablicaKomunikatowZnacznikZapisu ,
						intTablicaKomunikatowRozmiar := intTablicaKomunikatowRozmiar ,
						sWyslanyKomunikat := sWyslanyKomunikatDummy);
			sDane := '';
		END_IF	
	END_IF	
	IF wAlarmsWord3 <> wAlarmsWord3Zaraportowana THEN
	wAlarmsWord3Zaraportowana := wAlarmsWord3;
	fnKomunikatDaneDodaj_xOverFlow(sDane := sDane , sAtrybut := 'ALARMWORD3=' , sWartosc := WORD_TO_STRING(wAlarmsWord3) , xOverFlow := xOverFlow);	
		IF xOverFlow = TRUE THEN
			fnZapiszKomunikat(	sCalyKomunikat := '' ,
						sTypKomunikatu := 'A' ,
						sMnemonik := sMnemonik ,
						sMACAdres := sMACAdres ,
						sIDNadawcy := sIdInstancji ,
						sIDOdbiorcy := sIdAplikacji ,
						sDaneZapasowe := sDaneZapasowe ,
						sDane := sDane ,
						arTablicaKomunikatow := arTablicaKomunikatow ,
						intTablicaKomunikatowZnacznikZapisu := intTablicaKomunikatowZnacznikZapisu ,
						intTablicaKomunikatowRozmiar := intTablicaKomunikatowRozmiar ,
						sWyslanyKomunikat := sWyslanyKomunikatDummy);
			sDane := '';
		END_IF	
	END_IF	
	IF wAlarmsWord4 <> wAlarmsWord4Zaraportowana THEN
	wAlarmsWord4Zaraportowana := wAlarmsWord4;
	fnKomunikatDaneDodaj_xOverFlow(sDane := sDane , sAtrybut := 'ALARMWORD4=' , sWartosc := WORD_TO_STRING(wAlarmsWord4) , xOverFlow := xOverFlow);	
		IF xOverFlow = TRUE THEN
			fnZapiszKomunikat(	sCalyKomunikat := '' ,
						sTypKomunikatu := 'A' ,
						sMnemonik := sMnemonik ,
						sMACAdres := sMACAdres ,
						sIDNadawcy := sIdInstancji ,
						sIDOdbiorcy := sIdAplikacji ,
						sDaneZapasowe := sDaneZapasowe ,
						sDane := sDane ,
						arTablicaKomunikatow := arTablicaKomunikatow ,
						intTablicaKomunikatowZnacznikZapisu := intTablicaKomunikatowZnacznikZapisu ,
						intTablicaKomunikatowRozmiar := intTablicaKomunikatowRozmiar ,
						sWyslanyKomunikat := sWyslanyKomunikatDummy);
			sDane := '';
		END_IF	
	END_IF	
	IF xInstalacjaHC1 OR xInstalacjaHC2 THEN
		IF rTemperaturaZewnetrzna <> rTemperaturaZewnetrznaZaraportowana AND arModbusStatusKomunikacji[bAdres] = enumModbusStatus.KomunikacjaPrawidlowa THEN
			rTemperaturaZewnetrznaZaraportowana := rTemperaturaZewnetrzna;
			fnKomunikatDaneDodaj_xOverFlow(sDane := sDane , sAtrybut := 'TEMPZEW=' , sWartosc := REAL_TO_STRING(rTemperaturaZewnetrzna) , xOverFlow := xOverFlow);	
			IF xOverFlow = TRUE THEN
				fnZapiszKomunikat(	sCalyKomunikat := '' ,
							sTypKomunikatu := 'A' ,
							sMnemonik := sMnemonik ,
							sMACAdres := sMACAdres ,
							sIDNadawcy := sIdInstancji ,
							sIDOdbiorcy := sIdAplikacji ,
							sDaneZapasowe := sDaneZapasowe ,
							sDane := sDane ,
							arTablicaKomunikatow := arTablicaKomunikatow ,
							intTablicaKomunikatowZnacznikZapisu := intTablicaKomunikatowZnacznikZapisu ,
							intTablicaKomunikatowRozmiar := intTablicaKomunikatowRozmiar ,
							sWyslanyKomunikat := sWyslanyKomunikatDummy);
				sDane := '';
			END_IF
		END_IF
	END_IF
	IF xInstalacjaHC1 THEN
		IF rTemperaturaGrzaniaNastawionaHC1 <> rTemperaturaGrzaniaNastawionaHC1Zaraportowana AND arModbusStatusKomunikacji[bAdres] = enumModbusStatus.KomunikacjaPrawidlowa THEN
			rTemperaturaGrzaniaNastawionaHC1Zaraportowana := rTemperaturaGrzaniaNastawionaHC1;
			fnKomunikatDaneDodaj_xOverFlow(sDane := sDane , sAtrybut := 'TEMPNASHC1=' , sWartosc := REAL_TO_STRING(rTemperaturaGrzaniaNastawionaHC1) , xOverFlow := xOverFlow);	
			IF xOverFlow = TRUE THEN
				fnZapiszKomunikat(	sCalyKomunikat := '' ,
							sTypKomunikatu := 'A' ,
							sMnemonik := sMnemonik ,
							sMACAdres := sMACAdres ,
							sIDNadawcy := sIdInstancji ,
							sIDOdbiorcy := sIdAplikacji ,
							sDaneZapasowe := sDaneZapasowe ,
							sDane := sDane ,
							arTablicaKomunikatow := arTablicaKomunikatow ,
							intTablicaKomunikatowZnacznikZapisu := intTablicaKomunikatowZnacznikZapisu ,
							intTablicaKomunikatowRozmiar := intTablicaKomunikatowRozmiar ,
							sWyslanyKomunikat := sWyslanyKomunikatDummy);
				sDane := '';
			END_IF
		END_IF
		IF rTemperaturaGrzaniaNastawionaKrzywaGrzewczaHC1 <> rTemperaturaGrzaniaNastawionaKrzywaGrzewczaHC1Zaraportowana AND arModbusStatusKomunikacji[bAdres] = enumModbusStatus.KomunikacjaPrawidlowa THEN
			rTemperaturaGrzaniaNastawionaKrzywaGrzewczaHC1Zaraportowana := rTemperaturaGrzaniaNastawionaKrzywaGrzewczaHC1;
			fnKomunikatDaneDodaj_xOverFlow(sDane := sDane , sAtrybut := 'TEMPNASKGHC1=' , sWartosc := REAL_TO_STRING(rTemperaturaGrzaniaNastawionaKrzywaGrzewczaHC1) , xOverFlow := xOverFlow);	
			IF xOverFlow = TRUE THEN
				fnZapiszKomunikat(	sCalyKomunikat := '' ,
							sTypKomunikatu := 'A' ,
							sMnemonik := sMnemonik ,
							sMACAdres := sMACAdres ,
							sIDNadawcy := sIdInstancji ,
							sIDOdbiorcy := sIdAplikacji ,
							sDaneZapasowe := sDaneZapasowe ,
							sDane := sDane ,
							arTablicaKomunikatow := arTablicaKomunikatow ,
							intTablicaKomunikatowZnacznikZapisu := intTablicaKomunikatowZnacznikZapisu ,
							intTablicaKomunikatowRozmiar := intTablicaKomunikatowRozmiar ,
							sWyslanyKomunikat := sWyslanyKomunikatDummy);
				sDane := '';
			END_IF
		END_IF
		IF intTrybPracyHC1 <> intTrybPracyHC1Zaraportowana AND arModbusStatusKomunikacji[bAdres] = enumModbusStatus.KomunikacjaPrawidlowa THEN
			intTrybPracyHC1Zaraportowana := intTrybPracyHC1;
			fnKomunikatDaneDodaj_xOverFlow(sDane := sDane , sAtrybut := 'TRYBNASHC1=' , sWartosc := INT_TO_STRING(intTrybPracyHC1) , xOverFlow := xOverFlow);	
			IF xOverFlow = TRUE THEN
				fnZapiszKomunikat(	sCalyKomunikat := '' ,
							sTypKomunikatu := 'A' ,
							sMnemonik := sMnemonik ,
							sMACAdres := sMACAdres ,
							sIDNadawcy := sIdInstancji ,
							sIDOdbiorcy := sIdAplikacji ,
							sDaneZapasowe := sDaneZapasowe ,
							sDane := sDane ,
							arTablicaKomunikatow := arTablicaKomunikatow ,
							intTablicaKomunikatowZnacznikZapisu := intTablicaKomunikatowZnacznikZapisu ,
							intTablicaKomunikatowRozmiar := intTablicaKomunikatowRozmiar ,
							sWyslanyKomunikat := sWyslanyKomunikatDummy);
				sDane := '';
			END_IF
		END_IF
		IF intTrybOperacjiHC1 <> intTrybOperacjiHC1Zaraportowana AND arModbusStatusKomunikacji[bAdres] = enumModbusStatus.KomunikacjaPrawidlowa THEN
			intTrybOperacjiHC1Zaraportowana := intTrybOperacjiHC1;
			fnKomunikatDaneDodaj_xOverFlow(sDane := sDane , sAtrybut := 'TRYBOPHC1=' , sWartosc := INT_TO_STRING(intTrybOperacjiHC1) , xOverFlow := xOverFlow);	
			IF xOverFlow = TRUE THEN
				fnZapiszKomunikat(	sCalyKomunikat := '' ,
							sTypKomunikatu := 'A' ,
							sMnemonik := sMnemonik ,
							sMACAdres := sMACAdres ,
							sIDNadawcy := sIdInstancji ,
							sIDOdbiorcy := sIdAplikacji ,
							sDaneZapasowe := sDaneZapasowe ,
							sDane := sDane ,
							arTablicaKomunikatow := arTablicaKomunikatow ,
							intTablicaKomunikatowZnacznikZapisu := intTablicaKomunikatowZnacznikZapisu ,
							intTablicaKomunikatowRozmiar := intTablicaKomunikatowRozmiar ,
							sWyslanyKomunikat := sWyslanyKomunikatDummy);
				sDane := '';
			END_IF
		END_IF
		IF rTemperaturaZasilaniaObwoduHC1 <> rTemperaturaZasilaniaObwoduHC1Zaraportowana AND arModbusStatusKomunikacji[bAdres] = enumModbusStatus.KomunikacjaPrawidlowa THEN
			rTemperaturaZasilaniaObwoduHC1Zaraportowana := rTemperaturaZasilaniaObwoduHC1;
			fnKomunikatDaneDodaj_xOverFlow(sDane := sDane , sAtrybut := 'TEMPZASOHC1=' , sWartosc := REAL_TO_STRING(rTemperaturaZasilaniaObwoduHC1) , xOverFlow := xOverFlow);	
			IF xOverFlow = TRUE THEN
				fnZapiszKomunikat(	sCalyKomunikat := '' ,
							sTypKomunikatu := 'A' ,
							sMnemonik := sMnemonik ,
							sMACAdres := sMACAdres ,
							sIDNadawcy := sIdInstancji ,
							sIDOdbiorcy := sIdAplikacji ,
							sDaneZapasowe := sDaneZapasowe ,
							sDane := sDane ,
							arTablicaKomunikatow := arTablicaKomunikatow ,
							intTablicaKomunikatowZnacznikZapisu := intTablicaKomunikatowZnacznikZapisu ,
							intTablicaKomunikatowRozmiar := intTablicaKomunikatowRozmiar ,
							sWyslanyKomunikat := sWyslanyKomunikatDummy);
				sDane := '';
			END_IF
		END_IF
		IF rTemperaturaPowrotuObwoduHC1 <> rTemperaturaPowrotuObwoduHC1Zaraportowana AND arModbusStatusKomunikacji[bAdres] = enumModbusStatus.KomunikacjaPrawidlowa THEN
			rTemperaturaPowrotuObwoduHC1Zaraportowana := rTemperaturaPowrotuObwoduHC1;
			fnKomunikatDaneDodaj_xOverFlow(sDane := sDane , sAtrybut := 'TEMPPOWOHC1=' , sWartosc := REAL_TO_STRING(rTemperaturaPowrotuObwoduHC1) , xOverFlow := xOverFlow);	
			IF xOverFlow = TRUE THEN
				fnZapiszKomunikat(	sCalyKomunikat := '' ,
							sTypKomunikatu := 'A' ,
							sMnemonik := sMnemonik ,
							sMACAdres := sMACAdres ,
							sIDNadawcy := sIdInstancji ,
							sIDOdbiorcy := sIdAplikacji ,
							sDaneZapasowe := sDaneZapasowe ,
							sDane := sDane ,
							arTablicaKomunikatow := arTablicaKomunikatow ,
							intTablicaKomunikatowZnacznikZapisu := intTablicaKomunikatowZnacznikZapisu ,
							intTablicaKomunikatowRozmiar := intTablicaKomunikatowRozmiar ,
							sWyslanyKomunikat := sWyslanyKomunikatDummy);
				sDane := '';
			END_IF
		END_IF
		IF rTemperaturaPowrotuMiastoHC1 <> rTemperaturaPowrotuMiastoHC1Zaraportowana AND arModbusStatusKomunikacji[bAdres] = enumModbusStatus.KomunikacjaPrawidlowa THEN
			rTemperaturaPowrotuMiastoHC1Zaraportowana := rTemperaturaPowrotuMiastoHC1;
			fnKomunikatDaneDodaj_xOverFlow(sDane := sDane , sAtrybut := 'TEMPPOWMHC1=' , sWartosc := REAL_TO_STRING(rTemperaturaPowrotuMiastoHC1) , xOverFlow := xOverFlow);	
			IF xOverFlow = TRUE THEN
				fnZapiszKomunikat(	sCalyKomunikat := '' ,
							sTypKomunikatu := 'A' ,
							sMnemonik := sMnemonik ,
							sMACAdres := sMACAdres ,
							sIDNadawcy := sIdInstancji ,
							sIDOdbiorcy := sIdAplikacji ,
							sDaneZapasowe := sDaneZapasowe ,
							sDane := sDane ,
							arTablicaKomunikatow := arTablicaKomunikatow ,
							intTablicaKomunikatowZnacznikZapisu := intTablicaKomunikatowZnacznikZapisu ,
							intTablicaKomunikatowRozmiar := intTablicaKomunikatowRozmiar ,
							sWyslanyKomunikat := sWyslanyKomunikatDummy);
				sDane := '';
			END_IF
		END_IF
		IF rTemperaturaZasilaniaBudynku <> rTemperaturaZasilaniaBudynkuZaraportowana AND arModbusStatusKomunikacji[bAdres] = enumModbusStatus.KomunikacjaPrawidlowa THEN
			rTemperaturaZasilaniaBudynkuZaraportowana := rTemperaturaZasilaniaBudynku;
			fnKomunikatDaneDodaj_xOverFlow(sDane := sDane , sAtrybut := 'TEMPZASB=' , sWartosc := REAL_TO_STRING(rTemperaturaZasilaniaBudynku) , xOverFlow := xOverFlow);	
			IF xOverFlow = TRUE THEN
				fnZapiszKomunikat(	sCalyKomunikat := '' ,
							sTypKomunikatu := 'A' ,
							sMnemonik := sMnemonik ,
							sMACAdres := sMACAdres ,
							sIDNadawcy := sIdInstancji ,
							sIDOdbiorcy := sIdAplikacji ,
							sDaneZapasowe := sDaneZapasowe ,
							sDane := sDane ,
							arTablicaKomunikatow := arTablicaKomunikatow ,
							intTablicaKomunikatowZnacznikZapisu := intTablicaKomunikatowZnacznikZapisu ,
							intTablicaKomunikatowRozmiar := intTablicaKomunikatowRozmiar ,
							sWyslanyKomunikat := sWyslanyKomunikatDummy);
				sDane := '';
			END_IF
		END_IF
		IF rTemperaturaPowrotuBudynku <> rTemperaturaPowrotuBudynkuZaraportowana AND arModbusStatusKomunikacji[bAdres] = enumModbusStatus.KomunikacjaPrawidlowa THEN
			rTemperaturaPowrotuBudynkuZaraportowana := rTemperaturaPowrotuBudynku;
			fnKomunikatDaneDodaj_xOverFlow(sDane := sDane , sAtrybut := 'TEMPPOWB=' , sWartosc := REAL_TO_STRING(rTemperaturaPowrotuBudynku) , xOverFlow := xOverFlow);	
			IF xOverFlow = TRUE THEN
				fnZapiszKomunikat(	sCalyKomunikat := '' ,
							sTypKomunikatu := 'A' ,
							sMnemonik := sMnemonik ,
							sMACAdres := sMACAdres ,
							sIDNadawcy := sIdInstancji ,
							sIDOdbiorcy := sIdAplikacji ,
							sDaneZapasowe := sDaneZapasowe ,
							sDane := sDane ,
							arTablicaKomunikatow := arTablicaKomunikatow ,
							intTablicaKomunikatowZnacznikZapisu := intTablicaKomunikatowZnacznikZapisu ,
							intTablicaKomunikatowRozmiar := intTablicaKomunikatowRozmiar ,
							sWyslanyKomunikat := sWyslanyKomunikatDummy);
				sDane := '';
			END_IF
		END_IF
		IF rSygnalZadaniaGrzaniaHC1 <> rSygnalZadaniaGrzaniaHC1Zaraportowana AND arModbusStatusKomunikacji[bAdres] = enumModbusStatus.KomunikacjaPrawidlowa THEN
			rSygnalZadaniaGrzaniaHC1Zaraportowana := rSygnalZadaniaGrzaniaHC1;
			fnKomunikatDaneDodaj_xOverFlow(sDane := sDane , sAtrybut := 'STERGRZHC1=' , sWartosc := REAL_TO_STRING(rSygnalZadaniaGrzaniaHC1) , xOverFlow := xOverFlow);	
			IF xOverFlow = TRUE THEN
				fnZapiszKomunikat(	sCalyKomunikat := '' ,
							sTypKomunikatu := 'A' ,
							sMnemonik := sMnemonik ,
							sMACAdres := sMACAdres ,
							sIDNadawcy := sIdInstancji ,
							sIDOdbiorcy := sIdAplikacji ,
							sDaneZapasowe := sDaneZapasowe ,
							sDane := sDane ,
							arTablicaKomunikatow := arTablicaKomunikatow ,
							intTablicaKomunikatowZnacznikZapisu := intTablicaKomunikatowZnacznikZapisu ,
							intTablicaKomunikatowRozmiar := intTablicaKomunikatowRozmiar ,
							sWyslanyKomunikat := sWyslanyKomunikatDummy);
				sDane := '';
			END_IF
		END_IF
		IF rStopienOtwarciaZaworuMiastoHC1 <> rStopienOtwarciaZaworuMiastoHC1Zaraportowana AND arModbusStatusKomunikacji[bAdres] = enumModbusStatus.KomunikacjaPrawidlowa THEN
			rStopienOtwarciaZaworuMiastoHC1Zaraportowana := rStopienOtwarciaZaworuMiastoHC1;
			fnKomunikatDaneDodaj_xOverFlow(sDane := sDane , sAtrybut := 'STERZAWMHC1=' , sWartosc := REAL_TO_STRING(rStopienOtwarciaZaworuMiastoHC1) , xOverFlow := xOverFlow);	
			IF xOverFlow = TRUE THEN
				fnZapiszKomunikat(	sCalyKomunikat := '' ,
							sTypKomunikatu := 'A' ,
							sMnemonik := sMnemonik ,
							sMACAdres := sMACAdres ,
							sIDNadawcy := sIdInstancji ,
							sIDOdbiorcy := sIdAplikacji ,
							sDaneZapasowe := sDaneZapasowe ,
							sDane := sDane ,
							arTablicaKomunikatow := arTablicaKomunikatow ,
							intTablicaKomunikatowZnacznikZapisu := intTablicaKomunikatowZnacznikZapisu ,
							intTablicaKomunikatowRozmiar := intTablicaKomunikatowRozmiar ,
							sWyslanyKomunikat := sWyslanyKomunikatDummy);
				sDane := '';
			END_IF
		END_IF
		IF rKrzywaGrzewczaTemperaturyZewnetrznejX2HC1 <> rKrzywaGrzewczaTemperaturyZewnetrznejX2HC1Zaraportowana AND arModbusStatusKomunikacji[bAdres] = enumModbusStatus.KomunikacjaPrawidlowa THEN
			rKrzywaGrzewczaTemperaturyZewnetrznejX2HC1Zaraportowana := rKrzywaGrzewczaTemperaturyZewnetrznejX2HC1;
			fnKomunikatDaneDodaj_xOverFlow(sDane := sDane , sAtrybut := 'TEMPKGHC1X2=' , sWartosc := REAL_TO_STRING(rKrzywaGrzewczaTemperaturyZewnetrznejX2HC1) , xOverFlow := xOverFlow);	
			IF xOverFlow = TRUE THEN
				fnZapiszKomunikat(	sCalyKomunikat := '' ,
							sTypKomunikatu := 'A' ,
							sMnemonik := sMnemonik ,
							sMACAdres := sMACAdres ,
							sIDNadawcy := sIdInstancji ,
							sIDOdbiorcy := sIdAplikacji ,
							sDaneZapasowe := sDaneZapasowe ,
							sDane := sDane ,
							arTablicaKomunikatow := arTablicaKomunikatow ,
							intTablicaKomunikatowZnacznikZapisu := intTablicaKomunikatowZnacznikZapisu ,
							intTablicaKomunikatowRozmiar := intTablicaKomunikatowRozmiar ,
							sWyslanyKomunikat := sWyslanyKomunikatDummy);
				sDane := '';
			END_IF
		END_IF
		IF rKrzywaGrzewczaTemperaturyZewnetrznejX3HC1 <> rKrzywaGrzewczaTemperaturyZewnetrznejX3HC1Zaraportowana AND arModbusStatusKomunikacji[bAdres] = enumModbusStatus.KomunikacjaPrawidlowa THEN
			rKrzywaGrzewczaTemperaturyZewnetrznejX3HC1Zaraportowana := rKrzywaGrzewczaTemperaturyZewnetrznejX3HC1;
			fnKomunikatDaneDodaj_xOverFlow(sDane := sDane , sAtrybut := 'TEMPKGHC1X3=' , sWartosc := REAL_TO_STRING(rKrzywaGrzewczaTemperaturyZewnetrznejX3HC1) , xOverFlow := xOverFlow);	
			IF xOverFlow = TRUE THEN
				fnZapiszKomunikat(	sCalyKomunikat := '' ,
							sTypKomunikatu := 'A' ,
							sMnemonik := sMnemonik ,
							sMACAdres := sMACAdres ,
							sIDNadawcy := sIdInstancji ,
							sIDOdbiorcy := sIdAplikacji ,
							sDaneZapasowe := sDaneZapasowe ,
							sDane := sDane ,
							arTablicaKomunikatow := arTablicaKomunikatow ,
							intTablicaKomunikatowZnacznikZapisu := intTablicaKomunikatowZnacznikZapisu ,
							intTablicaKomunikatowRozmiar := intTablicaKomunikatowRozmiar ,
							sWyslanyKomunikat := sWyslanyKomunikatDummy);
				sDane := '';
			END_IF
		END_IF
		IF rKrzywaGrzewczaTemperaturyZewnetrznejX4HC1 <> rKrzywaGrzewczaTemperaturyZewnetrznejX4HC1Zaraportowana AND arModbusStatusKomunikacji[bAdres] = enumModbusStatus.KomunikacjaPrawidlowa THEN
			rKrzywaGrzewczaTemperaturyZewnetrznejX4HC1Zaraportowana := rKrzywaGrzewczaTemperaturyZewnetrznejX4HC1;
			fnKomunikatDaneDodaj_xOverFlow(sDane := sDane , sAtrybut := 'TEMPKGHC1X4=' , sWartosc := REAL_TO_STRING(rKrzywaGrzewczaTemperaturyZewnetrznejX4HC1) , xOverFlow := xOverFlow);	
			IF xOverFlow = TRUE THEN
				fnZapiszKomunikat(	sCalyKomunikat := '' ,
							sTypKomunikatu := 'A' ,
							sMnemonik := sMnemonik ,
							sMACAdres := sMACAdres ,
							sIDNadawcy := sIdInstancji ,
							sIDOdbiorcy := sIdAplikacji ,
							sDaneZapasowe := sDaneZapasowe ,
							sDane := sDane ,
							arTablicaKomunikatow := arTablicaKomunikatow ,
							intTablicaKomunikatowZnacznikZapisu := intTablicaKomunikatowZnacznikZapisu ,
							intTablicaKomunikatowRozmiar := intTablicaKomunikatowRozmiar ,
							sWyslanyKomunikat := sWyslanyKomunikatDummy);
				sDane := '';
			END_IF
		END_IF
		IF rKrzywaGrzewczaTemperaturyZewnetrznejX5HC1 <> rKrzywaGrzewczaTemperaturyZewnetrznejX5HC1Zaraportowana AND arModbusStatusKomunikacji[bAdres] = enumModbusStatus.KomunikacjaPrawidlowa THEN
			rKrzywaGrzewczaTemperaturyZewnetrznejX5HC1Zaraportowana := rKrzywaGrzewczaTemperaturyZewnetrznejX5HC1;
			fnKomunikatDaneDodaj_xOverFlow(sDane := sDane , sAtrybut := 'TEMPKGHC1X5=' , sWartosc := REAL_TO_STRING(rKrzywaGrzewczaTemperaturyZewnetrznejX5HC1) , xOverFlow := xOverFlow);	
			IF xOverFlow = TRUE THEN
				fnZapiszKomunikat(	sCalyKomunikat := '' ,
							sTypKomunikatu := 'A' ,
							sMnemonik := sMnemonik ,
							sMACAdres := sMACAdres ,
							sIDNadawcy := sIdInstancji ,
							sIDOdbiorcy := sIdAplikacji ,
							sDaneZapasowe := sDaneZapasowe ,
							sDane := sDane ,
							arTablicaKomunikatow := arTablicaKomunikatow ,
							intTablicaKomunikatowZnacznikZapisu := intTablicaKomunikatowZnacznikZapisu ,
							intTablicaKomunikatowRozmiar := intTablicaKomunikatowRozmiar ,
							sWyslanyKomunikat := sWyslanyKomunikatDummy);
				sDane := '';
			END_IF
		END_IF
		IF rKrzywaGrzewczaTemperaturyZewnetrznejX6HC1 <> rKrzywaGrzewczaTemperaturyZewnetrznejX6HC1Zaraportowana AND arModbusStatusKomunikacji[bAdres] = enumModbusStatus.KomunikacjaPrawidlowa THEN
			rKrzywaGrzewczaTemperaturyZewnetrznejX6HC1Zaraportowana := rKrzywaGrzewczaTemperaturyZewnetrznejX6HC1;
			fnKomunikatDaneDodaj_xOverFlow(sDane := sDane , sAtrybut := 'TEMPKGHC1X6=' , sWartosc := REAL_TO_STRING(rKrzywaGrzewczaTemperaturyZewnetrznejX6HC1) , xOverFlow := xOverFlow);	
			IF xOverFlow = TRUE THEN
				fnZapiszKomunikat(	sCalyKomunikat := '' ,
							sTypKomunikatu := 'A' ,
							sMnemonik := sMnemonik ,
							sMACAdres := sMACAdres ,
							sIDNadawcy := sIdInstancji ,
							sIDOdbiorcy := sIdAplikacji ,
							sDaneZapasowe := sDaneZapasowe ,
							sDane := sDane ,
							arTablicaKomunikatow := arTablicaKomunikatow ,
							intTablicaKomunikatowZnacznikZapisu := intTablicaKomunikatowZnacznikZapisu ,
							intTablicaKomunikatowRozmiar := intTablicaKomunikatowRozmiar ,
							sWyslanyKomunikat := sWyslanyKomunikatDummy);
				sDane := '';
			END_IF
		END_IF
		IF rKrzywaGrzewczaTemperaturyZasilaniaY2HC1 <> rKrzywaGrzewczaTemperaturyZasilaniaY2HC1Zaraportowana AND arModbusStatusKomunikacji[bAdres] = enumModbusStatus.KomunikacjaPrawidlowa THEN
			rKrzywaGrzewczaTemperaturyZasilaniaY2HC1Zaraportowana := rKrzywaGrzewczaTemperaturyZasilaniaY2HC1;
			fnKomunikatDaneDodaj_xOverFlow(sDane := sDane , sAtrybut := 'TEMPKGHC1Y2=' , sWartosc := REAL_TO_STRING(rKrzywaGrzewczaTemperaturyZasilaniaY2HC1) , xOverFlow := xOverFlow);	
			IF xOverFlow = TRUE THEN
				fnZapiszKomunikat(	sCalyKomunikat := '' ,
							sTypKomunikatu := 'A' ,
							sMnemonik := sMnemonik ,
							sMACAdres := sMACAdres ,
							sIDNadawcy := sIdInstancji ,
							sIDOdbiorcy := sIdAplikacji ,
							sDaneZapasowe := sDaneZapasowe ,
							sDane := sDane ,
							arTablicaKomunikatow := arTablicaKomunikatow ,
							intTablicaKomunikatowZnacznikZapisu := intTablicaKomunikatowZnacznikZapisu ,
							intTablicaKomunikatowRozmiar := intTablicaKomunikatowRozmiar ,
							sWyslanyKomunikat := sWyslanyKomunikatDummy);
				sDane := '';
			END_IF
		END_IF
		IF rKrzywaGrzewczaTemperaturyZasilaniaY3HC1 <> rKrzywaGrzewczaTemperaturyZasilaniaY3HC1Zaraportowana AND arModbusStatusKomunikacji[bAdres] = enumModbusStatus.KomunikacjaPrawidlowa THEN
			rKrzywaGrzewczaTemperaturyZasilaniaY3HC1Zaraportowana := rKrzywaGrzewczaTemperaturyZasilaniaY3HC1;
			fnKomunikatDaneDodaj_xOverFlow(sDane := sDane , sAtrybut := 'TEMPKGHC1Y3=' , sWartosc := REAL_TO_STRING(rKrzywaGrzewczaTemperaturyZasilaniaY3HC1) , xOverFlow := xOverFlow);	
			IF xOverFlow = TRUE THEN
				fnZapiszKomunikat(	sCalyKomunikat := '' ,
							sTypKomunikatu := 'A' ,
							sMnemonik := sMnemonik ,
							sMACAdres := sMACAdres ,
							sIDNadawcy := sIdInstancji ,
							sIDOdbiorcy := sIdAplikacji ,
							sDaneZapasowe := sDaneZapasowe ,
							sDane := sDane ,
							arTablicaKomunikatow := arTablicaKomunikatow ,
							intTablicaKomunikatowZnacznikZapisu := intTablicaKomunikatowZnacznikZapisu ,
							intTablicaKomunikatowRozmiar := intTablicaKomunikatowRozmiar ,
							sWyslanyKomunikat := sWyslanyKomunikatDummy);
				sDane := '';
			END_IF
		END_IF
		IF rKrzywaGrzewczaTemperaturyZasilaniaY4HC1 <> rKrzywaGrzewczaTemperaturyZasilaniaY4HC1Zaraportowana AND arModbusStatusKomunikacji[bAdres] = enumModbusStatus.KomunikacjaPrawidlowa THEN
			rKrzywaGrzewczaTemperaturyZasilaniaY4HC1Zaraportowana := rKrzywaGrzewczaTemperaturyZasilaniaY4HC1;
			fnKomunikatDaneDodaj_xOverFlow(sDane := sDane , sAtrybut := 'TEMPKGHC1Y4=' , sWartosc := REAL_TO_STRING(rKrzywaGrzewczaTemperaturyZasilaniaY4HC1) , xOverFlow := xOverFlow);	
			IF xOverFlow = TRUE THEN
				fnZapiszKomunikat(	sCalyKomunikat := '' ,
							sTypKomunikatu := 'A' ,
							sMnemonik := sMnemonik ,
							sMACAdres := sMACAdres ,
							sIDNadawcy := sIdInstancji ,
							sIDOdbiorcy := sIdAplikacji ,
							sDaneZapasowe := sDaneZapasowe ,
							sDane := sDane ,
							arTablicaKomunikatow := arTablicaKomunikatow ,
							intTablicaKomunikatowZnacznikZapisu := intTablicaKomunikatowZnacznikZapisu ,
							intTablicaKomunikatowRozmiar := intTablicaKomunikatowRozmiar ,
							sWyslanyKomunikat := sWyslanyKomunikatDummy);
				sDane := '';
			END_IF
		END_IF
		IF rKrzywaGrzewczaTemperaturyZasilaniaY5HC1 <> rKrzywaGrzewczaTemperaturyZasilaniaY5HC1Zaraportowana AND arModbusStatusKomunikacji[bAdres] = enumModbusStatus.KomunikacjaPrawidlowa THEN
			rKrzywaGrzewczaTemperaturyZasilaniaY5HC1Zaraportowana := rKrzywaGrzewczaTemperaturyZasilaniaY5HC1;
			fnKomunikatDaneDodaj_xOverFlow(sDane := sDane , sAtrybut := 'TEMPKGHC1Y5=' , sWartosc := REAL_TO_STRING(rKrzywaGrzewczaTemperaturyZasilaniaY5HC1) , xOverFlow := xOverFlow);	
			IF xOverFlow = TRUE THEN
				fnZapiszKomunikat(	sCalyKomunikat := '' ,
							sTypKomunikatu := 'A' ,
							sMnemonik := sMnemonik ,
							sMACAdres := sMACAdres ,
							sIDNadawcy := sIdInstancji ,
							sIDOdbiorcy := sIdAplikacji ,
							sDaneZapasowe := sDaneZapasowe ,
							sDane := sDane ,
							arTablicaKomunikatow := arTablicaKomunikatow ,
							intTablicaKomunikatowZnacznikZapisu := intTablicaKomunikatowZnacznikZapisu ,
							intTablicaKomunikatowRozmiar := intTablicaKomunikatowRozmiar ,
							sWyslanyKomunikat := sWyslanyKomunikatDummy);
				sDane := '';
			END_IF
		END_IF
		IF rKrzywaGrzewczaTemperaturyZasilaniaY6HC1 <> rKrzywaGrzewczaTemperaturyZasilaniaY6HC1Zaraportowana AND arModbusStatusKomunikacji[bAdres] = enumModbusStatus.KomunikacjaPrawidlowa THEN
			rKrzywaGrzewczaTemperaturyZasilaniaY6HC1Zaraportowana := rKrzywaGrzewczaTemperaturyZasilaniaY6HC1;
			fnKomunikatDaneDodaj_xOverFlow(sDane := sDane , sAtrybut := 'TEMPKGHC1Y6=' , sWartosc := REAL_TO_STRING(rKrzywaGrzewczaTemperaturyZasilaniaY6HC1) , xOverFlow := xOverFlow);	
			IF xOverFlow = TRUE THEN
				fnZapiszKomunikat(	sCalyKomunikat := '' ,
							sTypKomunikatu := 'A' ,
							sMnemonik := sMnemonik ,
							sMACAdres := sMACAdres ,
							sIDNadawcy := sIdInstancji ,
							sIDOdbiorcy := sIdAplikacji ,
							sDaneZapasowe := sDaneZapasowe ,
							sDane := sDane ,
							arTablicaKomunikatow := arTablicaKomunikatow ,
							intTablicaKomunikatowZnacznikZapisu := intTablicaKomunikatowZnacznikZapisu ,
							intTablicaKomunikatowRozmiar := intTablicaKomunikatowRozmiar ,
							sWyslanyKomunikat := sWyslanyKomunikatDummy);
				sDane := '';
			END_IF
		END_IF
		IF xSezonGrzewczy <> xSezonGrzewczyZaraportowana THEN
			xSezonGrzewczyZaraportowana := xSezonGrzewczy;
			fnKomunikatDaneDodaj_xOverFlow(sDane := sDane , sAtrybut := 'SEZONGRZ=' , sWartosc := BOOL_TO_STRING(xSezonGrzewczy) , xOverFlow := xOverFlow);	
			IF xOverFlow = TRUE THEN
				fnZapiszKomunikat(	sCalyKomunikat := '' ,
							sTypKomunikatu := 'M' ,
							sMnemonik := sMnemonik ,
							sMACAdres := sMACAdres ,
							sIDNadawcy := sIdInstancji ,
							sIDOdbiorcy := sIdAplikacji ,
							sDaneZapasowe := sDaneZapasowe ,
							sDane := sDane ,
							arTablicaKomunikatow := arTablicaKomunikatow ,
							intTablicaKomunikatowZnacznikZapisu := intTablicaKomunikatowZnacznikZapisu ,
							intTablicaKomunikatowRozmiar := intTablicaKomunikatowRozmiar ,
							sWyslanyKomunikat := sWyslanyKomunikatDummy);
				sDane := '';
			END_IF	
		END_IF	
		IF rTemperaturaSrednia1Dzien <> rTemperaturaSrednia1DzienZaraportowana THEN
			rTemperaturaSrednia1DzienZaraportowana := rTemperaturaSrednia1Dzien;
			fnKomunikatDaneDodaj_xOverFlow(sDane := sDane , sAtrybut := 'TEMPSR1DZ=' , sWartosc := REAL_TO_STRING(rTemperaturaSrednia1Dzien + 273.15) , xOverFlow := xOverFlow);	
			IF xOverFlow = TRUE THEN
				fnZapiszKomunikat(	sCalyKomunikat := '' ,
							sTypKomunikatu := 'M' ,
							sMnemonik := sMnemonik ,
							sMACAdres := sMACAdres ,
							sIDNadawcy := sIdInstancji ,
							sIDOdbiorcy := sIdAplikacji ,
							sDaneZapasowe := sDaneZapasowe ,
							sDane := sDane ,
							arTablicaKomunikatow := arTablicaKomunikatow ,
							intTablicaKomunikatowZnacznikZapisu := intTablicaKomunikatowZnacznikZapisu ,
							intTablicaKomunikatowRozmiar := intTablicaKomunikatowRozmiar ,
							sWyslanyKomunikat := sWyslanyKomunikatDummy);
				sDane := '';
			END_IF	
		END_IF	
	END_IF
	IF xInstalacjaDHW THEN
		IF rTemperaturaGrzaniaNastawionaDHW <> rTemperaturaGrzaniaNastawionaDHWZaraportowana AND arModbusStatusKomunikacji[bAdres] = enumModbusStatus.KomunikacjaPrawidlowa THEN
			rTemperaturaGrzaniaNastawionaDHWZaraportowana := rTemperaturaGrzaniaNastawionaDHW;
			fnKomunikatDaneDodaj_xOverFlow(sDane := sDane , sAtrybut := 'TEMPNASDHW=' , sWartosc := REAL_TO_STRING(rTemperaturaGrzaniaNastawionaDHW) , xOverFlow := xOverFlow);	
			IF xOverFlow = TRUE THEN
				fnZapiszKomunikat(	sCalyKomunikat := '' ,
							sTypKomunikatu := 'A' ,
							sMnemonik := sMnemonik ,
							sMACAdres := sMACAdres ,
							sIDNadawcy := sIdInstancji ,
							sIDOdbiorcy := sIdAplikacji ,
							sDaneZapasowe := sDaneZapasowe ,
							sDane := sDane ,
							arTablicaKomunikatow := arTablicaKomunikatow ,
							intTablicaKomunikatowZnacznikZapisu := intTablicaKomunikatowZnacznikZapisu ,
							intTablicaKomunikatowRozmiar := intTablicaKomunikatowRozmiar ,
							sWyslanyKomunikat := sWyslanyKomunikatDummy);
				sDane := '';
			END_IF
		END_IF
		IF intTrybPracyDHW <> intTrybPracyDHWZaraportowana AND arModbusStatusKomunikacji[bAdres] = enumModbusStatus.KomunikacjaPrawidlowa THEN
			intTrybPracyDHWZaraportowana := intTrybPracyDHW;
			fnKomunikatDaneDodaj_xOverFlow(sDane := sDane , sAtrybut := 'TRYBNASDHW=' , sWartosc := INT_TO_STRING(intTrybPracyDHW) , xOverFlow := xOverFlow);	
			IF xOverFlow = TRUE THEN
				fnZapiszKomunikat(	sCalyKomunikat := '' ,
							sTypKomunikatu := 'A' ,
							sMnemonik := sMnemonik ,
							sMACAdres := sMACAdres ,
							sIDNadawcy := sIdInstancji ,
							sIDOdbiorcy := sIdAplikacji ,
							sDaneZapasowe := sDaneZapasowe ,
							sDane := sDane ,
							arTablicaKomunikatow := arTablicaKomunikatow ,
							intTablicaKomunikatowZnacznikZapisu := intTablicaKomunikatowZnacznikZapisu ,
							intTablicaKomunikatowRozmiar := intTablicaKomunikatowRozmiar ,
							sWyslanyKomunikat := sWyslanyKomunikatDummy);
				sDane := '';
			END_IF
		END_IF
		IF intTrybOperacjiDHW <> intTrybOperacjiDHWZaraportowana AND arModbusStatusKomunikacji[bAdres] = enumModbusStatus.KomunikacjaPrawidlowa THEN
			intTrybOperacjiDHWZaraportowana := intTrybOperacjiDHW;
			fnKomunikatDaneDodaj_xOverFlow(sDane := sDane , sAtrybut := 'TRYBOPDHW=' , sWartosc := INT_TO_STRING(intTrybOperacjiDHW) , xOverFlow := xOverFlow);	
			IF xOverFlow = TRUE THEN
				fnZapiszKomunikat(	sCalyKomunikat := '' ,
							sTypKomunikatu := 'A' ,
							sMnemonik := sMnemonik ,
							sMACAdres := sMACAdres ,
							sIDNadawcy := sIdInstancji ,
							sIDOdbiorcy := sIdAplikacji ,
							sDaneZapasowe := sDaneZapasowe ,
							sDane := sDane ,
							arTablicaKomunikatow := arTablicaKomunikatow ,
							intTablicaKomunikatowZnacznikZapisu := intTablicaKomunikatowZnacznikZapisu ,
							intTablicaKomunikatowRozmiar := intTablicaKomunikatowRozmiar ,
							sWyslanyKomunikat := sWyslanyKomunikatDummy);
				sDane := '';
			END_IF
		END_IF
		IF rTemperaturaPowrotuMiastoDHW <> rTemperaturaPowrotuMiastoDHWZaraportowana AND arModbusStatusKomunikacji[bAdres] = enumModbusStatus.KomunikacjaPrawidlowa THEN
			rTemperaturaPowrotuMiastoDHWZaraportowana := rTemperaturaPowrotuMiastoDHW;
			fnKomunikatDaneDodaj_xOverFlow(sDane := sDane , sAtrybut := 'TEMPPOWMDHW=' , sWartosc := REAL_TO_STRING(rTemperaturaPowrotuMiastoDHW) , xOverFlow := xOverFlow);	
			IF xOverFlow = TRUE THEN
				fnZapiszKomunikat(	sCalyKomunikat := '' ,
							sTypKomunikatu := 'A' ,
							sMnemonik := sMnemonik ,
							sMACAdres := sMACAdres ,
							sIDNadawcy := sIdInstancji ,
							sIDOdbiorcy := sIdAplikacji ,
							sDaneZapasowe := sDaneZapasowe ,
							sDane := sDane ,
							arTablicaKomunikatow := arTablicaKomunikatow ,
							intTablicaKomunikatowZnacznikZapisu := intTablicaKomunikatowZnacznikZapisu ,
							intTablicaKomunikatowRozmiar := intTablicaKomunikatowRozmiar ,
							sWyslanyKomunikat := sWyslanyKomunikatDummy);
				sDane := '';
			END_IF
		END_IF
		IF rTemperaturaZasilaniaBudynekDHW <> rTemperaturaZasilaniaBudynekDHWZaraportowana AND arModbusStatusKomunikacji[bAdres] = enumModbusStatus.KomunikacjaPrawidlowa THEN
			rTemperaturaZasilaniaBudynekDHWZaraportowana := rTemperaturaZasilaniaBudynekDHW;
			fnKomunikatDaneDodaj_xOverFlow(sDane := sDane , sAtrybut := 'TEMPZASBDHW=' , sWartosc := REAL_TO_STRING(rTemperaturaZasilaniaBudynekDHW) , xOverFlow := xOverFlow);	
			IF xOverFlow = TRUE THEN
				fnZapiszKomunikat(	sCalyKomunikat := '' ,
							sTypKomunikatu := 'A' ,
							sMnemonik := sMnemonik ,
							sMACAdres := sMACAdres ,
							sIDNadawcy := sIdInstancji ,
							sIDOdbiorcy := sIdAplikacji ,
							sDaneZapasowe := sDaneZapasowe ,
							sDane := sDane ,
							arTablicaKomunikatow := arTablicaKomunikatow ,
							intTablicaKomunikatowZnacznikZapisu := intTablicaKomunikatowZnacznikZapisu ,
							intTablicaKomunikatowRozmiar := intTablicaKomunikatowRozmiar ,
							sWyslanyKomunikat := sWyslanyKomunikatDummy);
				sDane := '';
			END_IF
		END_IF
		IF rTemperaturaPowrotuBudynekDHW <> rTemperaturaPowrotuBudynekDHWZaraportowana AND arModbusStatusKomunikacji[bAdres] = enumModbusStatus.KomunikacjaPrawidlowa THEN
			rTemperaturaPowrotuBudynekDHWZaraportowana := rTemperaturaPowrotuBudynekDHW;
			fnKomunikatDaneDodaj_xOverFlow(sDane := sDane , sAtrybut := 'TEMPPOWBDHW=' , sWartosc := REAL_TO_STRING(rTemperaturaPowrotuBudynekDHW) , xOverFlow := xOverFlow);	
			IF xOverFlow = TRUE THEN
				fnZapiszKomunikat(	sCalyKomunikat := '' ,
							sTypKomunikatu := 'A' ,
							sMnemonik := sMnemonik ,
							sMACAdres := sMACAdres ,
							sIDNadawcy := sIdInstancji ,
							sIDOdbiorcy := sIdAplikacji ,
							sDaneZapasowe := sDaneZapasowe ,
							sDane := sDane ,
							arTablicaKomunikatow := arTablicaKomunikatow ,
							intTablicaKomunikatowZnacznikZapisu := intTablicaKomunikatowZnacznikZapisu ,
							intTablicaKomunikatowRozmiar := intTablicaKomunikatowRozmiar ,
							sWyslanyKomunikat := sWyslanyKomunikatDummy);
				sDane := '';
			END_IF
		END_IF
		IF rStopienOtwarciaZaworuMiastoDHW <> rStopienOtwarciaZaworuMiastoDHWZaraportowana AND arModbusStatusKomunikacji[bAdres] = enumModbusStatus.KomunikacjaPrawidlowa THEN
			rStopienOtwarciaZaworuMiastoDHWZaraportowana := rStopienOtwarciaZaworuMiastoDHW;
			fnKomunikatDaneDodaj_xOverFlow(sDane := sDane , sAtrybut := 'STERZAWMDHW=' , sWartosc := REAL_TO_STRING(rStopienOtwarciaZaworuMiastoDHW) , xOverFlow := xOverFlow);	
			IF xOverFlow = TRUE THEN
				fnZapiszKomunikat(	sCalyKomunikat := '' ,
							sTypKomunikatu := 'A' ,
							sMnemonik := sMnemonik ,
							sMACAdres := sMACAdres ,
							sIDNadawcy := sIdInstancji ,
							sIDOdbiorcy := sIdAplikacji ,
							sDaneZapasowe := sDaneZapasowe ,
							sDane := sDane ,
							arTablicaKomunikatow := arTablicaKomunikatow ,
							intTablicaKomunikatowZnacznikZapisu := intTablicaKomunikatowZnacznikZapisu ,
							intTablicaKomunikatowRozmiar := intTablicaKomunikatowRozmiar ,
							sWyslanyKomunikat := sWyslanyKomunikatDummy);
				sDane := '';
			END_IF
		END_IF
	END_IF
	IF sDane <> '' AND xPoInicjalizacji THEN
		fnZapiszKomunikat(	sCalyKomunikat := '' ,
							sTypKomunikatu := 'M' ,
							sMnemonik := sMnemonik ,
							sMACAdres := sMACAdres ,
							sIDNadawcy := sIdInstancji ,
							sIDOdbiorcy := sIdAplikacji ,
							sDaneZapasowe := sDaneZapasowe ,
							sDane := sDane ,
							arTablicaKomunikatow := arTablicaKomunikatow ,
							intTablicaKomunikatowZnacznikZapisu := intTablicaKomunikatowZnacznikZapisu ,
							intTablicaKomunikatowRozmiar := intTablicaKomunikatowRozmiar ,
							sWyslanyKomunikat := sWyslanyKomunikatDummy);
	END_IF
END_IF
	
// Obsługa alarmów do węzła ciepła
// Alarm komunikacji
IF arErrorStan[enumPPPSWezelClimatixPOL63xError.BrakKomunikacji] <> enumAlarmWartosc.StanAlarmowy AND arModbusStatusKomunikacji[bAdres] = enumModbusStatus.BrakKomunikacji THEN
	arErrorStan[enumPPPSWezelClimatixPOL63xError.BrakKomunikacji] := enumAlarmWartosc.StanAlarmowy;
	arErrorKlasa[enumPPPSWezelClimatixPOL63xError.BrakKomunikacji] := enumPPPSWezelClimatixPOL63xErrorKlasa.BrakKomunikacji;
	xBrakKomunikacji := TRUE;
	IF xPoInicjalizacji THEN
		fnZapiszKomunikat(	sCalyKomunikat := '' ,
							sTypKomunikatu := 'E' ,
							sMnemonik := sMnemonik ,
							sMACAdres := sMACAdres ,
							sIDNadawcy := sIdInstancji ,
							sIDOdbiorcy := sIdAplikacji ,
							sDaneZapasowe := sDaneZapasowe ,
							sDane := fnKomunikatDaneError(xAktywny := TRUE , intKlasa := enumPPPSWezelClimatixPOL63xErrorKlasa.BrakKomunikacji , intNumer := enumPPPSWezelClimatixPOL63xError.BrakKomunikacji),
							arTablicaKomunikatow := arTablicaKomunikatow ,
							intTablicaKomunikatowZnacznikZapisu := intTablicaKomunikatowZnacznikZapisu ,
							intTablicaKomunikatowRozmiar := intTablicaKomunikatowRozmiar ,
							sWyslanyKomunikat := sWyslanyKomunikatDummy);
	END_IF
END_IF
IF arErrorStan[enumPPPSWezelClimatixPOL63xError.BrakKomunikacji] <> enumAlarmWartosc.StanNormalny AND arModbusStatusKomunikacji[bAdres] = enumModbusStatus.KomunikacjaPrawidlowa THEN
	arErrorStan[enumPPPSWezelClimatixPOL63xError.BrakKomunikacji] := enumAlarmWartosc.StanNormalny;
	arErrorKlasa[enumPPPSWezelClimatixPOL63xError.BrakKomunikacji] := enumPPPSWezelClimatixPOL63xErrorKlasa.BrakKomunikacji;
	xBrakKomunikacji := FALSE;
	IF xPoInicjalizacji THEN
		fnZapiszKomunikat(	sCalyKomunikat := '' ,
							sTypKomunikatu := 'E' ,
							sMnemonik := sMnemonik ,
							sMACAdres := sMACAdres ,
							sIDNadawcy := sIdInstancji ,
							sIDOdbiorcy := sIdAplikacji ,
							sDaneZapasowe := sDaneZapasowe ,
							sDane := fnKomunikatDaneError(xAktywny := FALSE , intKlasa := enumPPPSWezelClimatixPOL63xErrorKlasa.BrakKomunikacji , intNumer := enumPPPSWezelClimatixPOL63xError.BrakKomunikacji),
							arTablicaKomunikatow := arTablicaKomunikatow ,
							intTablicaKomunikatowZnacznikZapisu := intTablicaKomunikatowZnacznikZapisu ,
							intTablicaKomunikatowRozmiar := intTablicaKomunikatowRozmiar ,
							sWyslanyKomunikat := sWyslanyKomunikatDummy);
	END_IF
END_IF
// Alarm ogólny w klasie bezpieczeństwa
IF arErrorStan[enumPPPSWezelClimatixPOL63xError.AlarmOgolnyBezpieczenstwa] <> enumAlarmWartosc.StanAlarmowy AND xOdczytanaKlasaAlarmuBezpieczenstwa AND arModbusStatusKomunikacji[bAdres] = enumModbusStatus.KomunikacjaPrawidlowa THEN
	arErrorStan[enumPPPSWezelClimatixPOL63xError.AlarmOgolnyBezpieczenstwa] := enumAlarmWartosc.StanAlarmowy;
	arErrorKlasa[enumPPPSWezelClimatixPOL63xError.AlarmOgolnyBezpieczenstwa] := enumPPPSWezelClimatixPOL63xErrorKlasa.AlarmOgolnyBezpieczenstwa;
	IF xPoInicjalizacji THEN
		fnZapiszKomunikat(	sCalyKomunikat := '' ,
							sTypKomunikatu := 'E' ,
							sMnemonik := sMnemonik ,
							sMACAdres := sMACAdres ,
							sIDNadawcy := sIdInstancji ,
							sIDOdbiorcy := sIdAplikacji ,
							sDaneZapasowe := sDaneZapasowe ,
							sDane := fnKomunikatDaneError(xAktywny := TRUE , intKlasa := enumPPPSWezelClimatixPOL63xErrorKlasa.AlarmOgolnyBezpieczenstwa , intNumer := enumPPPSWezelClimatixPOL63xError.AlarmOgolnyBezpieczenstwa),
							arTablicaKomunikatow := arTablicaKomunikatow ,
							intTablicaKomunikatowZnacznikZapisu := intTablicaKomunikatowZnacznikZapisu ,
							intTablicaKomunikatowRozmiar := intTablicaKomunikatowRozmiar ,
							sWyslanyKomunikat := sWyslanyKomunikatDummy);
	END_IF
END_IF
IF arErrorStan[enumPPPSWezelClimatixPOL63xError.AlarmOgolnyBezpieczenstwa] <> enumAlarmWartosc.StanNormalny AND NOT xOdczytanaKlasaAlarmuBezpieczenstwa AND arModbusStatusKomunikacji[bAdres] = enumModbusStatus.KomunikacjaPrawidlowa THEN
	arErrorStan[enumPPPSWezelClimatixPOL63xError.AlarmOgolnyBezpieczenstwa] := enumAlarmWartosc.StanNormalny;
	arErrorKlasa[enumPPPSWezelClimatixPOL63xError.AlarmOgolnyBezpieczenstwa] := enumPPPSWezelClimatixPOL63xErrorKlasa.AlarmOgolnyBezpieczenstwa;
	IF xPoInicjalizacji THEN
		fnZapiszKomunikat(	sCalyKomunikat := '' ,
							sTypKomunikatu := 'E' ,
							sMnemonik := sMnemonik ,
							sMACAdres := sMACAdres ,
							sIDNadawcy := sIdInstancji ,
							sIDOdbiorcy := sIdAplikacji ,
							sDaneZapasowe := sDaneZapasowe ,
							sDane := fnKomunikatDaneError(xAktywny := FALSE , intKlasa := enumPPPSWezelClimatixPOL63xErrorKlasa.AlarmOgolnyBezpieczenstwa , intNumer := enumPPPSWezelClimatixPOL63xError.AlarmOgolnyBezpieczenstwa),
							arTablicaKomunikatow := arTablicaKomunikatow ,
							intTablicaKomunikatowZnacznikZapisu := intTablicaKomunikatowZnacznikZapisu ,
							intTablicaKomunikatowRozmiar := intTablicaKomunikatowRozmiar ,
							sWyslanyKomunikat := sWyslanyKomunikatDummy);
	END_IF
END_IF
// Alarm ogólny w klasie krytycznej
IF arErrorStan[enumPPPSWezelClimatixPOL63xError.AlarmOgolnyKrytyczny] <> enumAlarmWartosc.StanAlarmowy AND xOdczytanaKlasaAlarmuKrytyczny AND arModbusStatusKomunikacji[bAdres] = enumModbusStatus.KomunikacjaPrawidlowa THEN
	arErrorStan[enumPPPSWezelClimatixPOL63xError.AlarmOgolnyKrytyczny] := enumAlarmWartosc.StanAlarmowy;
	arErrorKlasa[enumPPPSWezelClimatixPOL63xError.AlarmOgolnyKrytyczny] := enumPPPSWezelClimatixPOL63xErrorKlasa.AlarmOgolnyKrytyczny;
	IF xPoInicjalizacji THEN
		fnZapiszKomunikat(	sCalyKomunikat := '' ,
							sTypKomunikatu := 'E' ,
							sMnemonik := sMnemonik ,
							sMACAdres := sMACAdres ,
							sIDNadawcy := sIdInstancji ,
							sIDOdbiorcy := sIdAplikacji ,
							sDaneZapasowe := sDaneZapasowe ,
							sDane := fnKomunikatDaneError(xAktywny := TRUE , intKlasa := enumPPPSWezelClimatixPOL63xErrorKlasa.AlarmOgolnyKrytyczny , intNumer := enumPPPSWezelClimatixPOL63xError.AlarmOgolnyKrytyczny),
							arTablicaKomunikatow := arTablicaKomunikatow ,
							intTablicaKomunikatowZnacznikZapisu := intTablicaKomunikatowZnacznikZapisu ,
							intTablicaKomunikatowRozmiar := intTablicaKomunikatowRozmiar ,
							sWyslanyKomunikat := sWyslanyKomunikatDummy);
	END_IF
END_IF
IF arErrorStan[enumPPPSWezelClimatixPOL63xError.AlarmOgolnyKrytyczny] <> enumAlarmWartosc.StanNormalny AND NOT xOdczytanaKlasaAlarmuKrytyczny AND arModbusStatusKomunikacji[bAdres] = enumModbusStatus.KomunikacjaPrawidlowa THEN
	arErrorStan[enumPPPSWezelClimatixPOL63xError.AlarmOgolnyKrytyczny] := enumAlarmWartosc.StanNormalny;
	arErrorKlasa[enumPPPSWezelClimatixPOL63xError.AlarmOgolnyKrytyczny] := enumPPPSWezelClimatixPOL63xErrorKlasa.AlarmOgolnyKrytyczny;
	IF xPoInicjalizacji THEN
		fnZapiszKomunikat(	sCalyKomunikat := '' ,
							sTypKomunikatu := 'E' ,
							sMnemonik := sMnemonik ,
							sMACAdres := sMACAdres ,
							sIDNadawcy := sIdInstancji ,
							sIDOdbiorcy := sIdAplikacji ,
							sDaneZapasowe := sDaneZapasowe ,
							sDane := fnKomunikatDaneError(xAktywny := FALSE , intKlasa := enumPPPSWezelClimatixPOL63xErrorKlasa.AlarmOgolnyKrytyczny , intNumer := enumPPPSWezelClimatixPOL63xError.AlarmOgolnyKrytyczny),
							arTablicaKomunikatow := arTablicaKomunikatow ,
							intTablicaKomunikatowZnacznikZapisu := intTablicaKomunikatowZnacznikZapisu ,
							intTablicaKomunikatowRozmiar := intTablicaKomunikatowRozmiar ,
							sWyslanyKomunikat := sWyslanyKomunikatDummy);
	END_IF
END_IF
// Alarm ogólny w klasie ostrzeżenia
IF arErrorStan[enumPPPSWezelClimatixPOL63xError.AlarmOgolnyOstrzezenie] <> enumAlarmWartosc.StanAlarmowy AND xOdczytanaKlasaAlarmuOstrzezenie AND arModbusStatusKomunikacji[bAdres] = enumModbusStatus.KomunikacjaPrawidlowa THEN
	arErrorStan[enumPPPSWezelClimatixPOL63xError.AlarmOgolnyOstrzezenie] := enumAlarmWartosc.StanAlarmowy;
	arErrorKlasa[enumPPPSWezelClimatixPOL63xError.AlarmOgolnyOstrzezenie] := enumPPPSWezelClimatixPOL63xErrorKlasa.AlarmOgolnyOstrzezenie;
	IF xPoInicjalizacji THEN
		fnZapiszKomunikat(	sCalyKomunikat := '' ,
							sTypKomunikatu := 'E' ,
							sMnemonik := sMnemonik ,
							sMACAdres := sMACAdres ,
							sIDNadawcy := sIdInstancji ,
							sIDOdbiorcy := sIdAplikacji ,
							sDaneZapasowe := sDaneZapasowe ,
							sDane := fnKomunikatDaneError(xAktywny := TRUE , intKlasa := enumPPPSWezelClimatixPOL63xErrorKlasa.AlarmOgolnyOstrzezenie , intNumer := enumPPPSWezelClimatixPOL63xError.AlarmOgolnyOstrzezenie),
							arTablicaKomunikatow := arTablicaKomunikatow ,
							intTablicaKomunikatowZnacznikZapisu := intTablicaKomunikatowZnacznikZapisu ,
							intTablicaKomunikatowRozmiar := intTablicaKomunikatowRozmiar ,
							sWyslanyKomunikat := sWyslanyKomunikatDummy);
	END_IF
END_IF
IF arErrorStan[enumPPPSWezelClimatixPOL63xError.AlarmOgolnyOstrzezenie] <> enumAlarmWartosc.StanNormalny AND NOT xOdczytanaKlasaAlarmuOstrzezenie AND arModbusStatusKomunikacji[bAdres] = enumModbusStatus.KomunikacjaPrawidlowa THEN
	arErrorStan[enumPPPSWezelClimatixPOL63xError.AlarmOgolnyOstrzezenie] := enumAlarmWartosc.StanNormalny;
	arErrorKlasa[enumPPPSWezelClimatixPOL63xError.AlarmOgolnyOstrzezenie] := enumPPPSWezelClimatixPOL63xErrorKlasa.AlarmOgolnyOstrzezenie;
	IF xPoInicjalizacji THEN
		fnZapiszKomunikat(	sCalyKomunikat := '' ,
							sTypKomunikatu := 'E' ,
							sMnemonik := sMnemonik ,
							sMACAdres := sMACAdres ,
							sIDNadawcy := sIdInstancji ,
							sIDOdbiorcy := sIdAplikacji ,
							sDaneZapasowe := sDaneZapasowe ,
							sDane := fnKomunikatDaneError(xAktywny := FALSE , intKlasa := enumPPPSWezelClimatixPOL63xErrorKlasa.AlarmOgolnyOstrzezenie , intNumer := enumPPPSWezelClimatixPOL63xError.AlarmOgolnyOstrzezenie),
							arTablicaKomunikatow := arTablicaKomunikatow ,
							intTablicaKomunikatowZnacznikZapisu := intTablicaKomunikatowZnacznikZapisu ,
							intTablicaKomunikatowRozmiar := intTablicaKomunikatowRozmiar ,
							sWyslanyKomunikat := sWyslanyKomunikatDummy);
	END_IF
END_IF
// Alarm czujnika zewnętrzengo
IF arErrorStan[enumPPPSWezelClimatixPOL63xError.AlarmCzujnikaZewnetrznego] <> enumAlarmWartosc.StanAlarmowy AND xBladBrakZmianyTemperaturyZewnetrznej AND arModbusStatusKomunikacji[bAdres] = enumModbusStatus.KomunikacjaPrawidlowa THEN
	arErrorStan[enumPPPSWezelClimatixPOL63xError.AlarmCzujnikaZewnetrznego] := enumAlarmWartosc.StanAlarmowy;
	arErrorKlasa[enumPPPSWezelClimatixPOL63xError.AlarmCzujnikaZewnetrznego] := enumPPPSWezelClimatixPOL63xErrorKlasa.AlarmCzujnikaZewnetrznego;
	IF xPoInicjalizacji THEN
		fnZapiszKomunikat(	sCalyKomunikat := '' ,
							sTypKomunikatu := 'E' ,
							sMnemonik := sMnemonik ,
							sMACAdres := sMACAdres ,
							sIDNadawcy := sIdInstancji ,
							sIDOdbiorcy := sIdAplikacji ,
							sDaneZapasowe := sDaneZapasowe ,
							sDane := fnKomunikatDaneError(xAktywny := TRUE , intKlasa := enumPPPSWezelClimatixPOL63xErrorKlasa.AlarmCzujnikaZewnetrznego , intNumer := enumPPPSWezelClimatixPOL63xError.AlarmCzujnikaZewnetrznego),
							arTablicaKomunikatow := arTablicaKomunikatow ,
							intTablicaKomunikatowZnacznikZapisu := intTablicaKomunikatowZnacznikZapisu ,
							intTablicaKomunikatowRozmiar := intTablicaKomunikatowRozmiar ,
							sWyslanyKomunikat := sWyslanyKomunikatDummy);
	END_IF
END_IF
IF arErrorStan[enumPPPSWezelClimatixPOL63xError.AlarmCzujnikaZewnetrznego] <> enumAlarmWartosc.StanNormalny AND NOT xBladBrakZmianyTemperaturyZewnetrznej AND arModbusStatusKomunikacji[bAdres] = enumModbusStatus.KomunikacjaPrawidlowa THEN
	arErrorStan[enumPPPSWezelClimatixPOL63xError.AlarmCzujnikaZewnetrznego] := enumAlarmWartosc.StanNormalny;
	arErrorKlasa[enumPPPSWezelClimatixPOL63xError.AlarmCzujnikaZewnetrznego] := enumPPPSWezelClimatixPOL63xErrorKlasa.AlarmCzujnikaZewnetrznego;
	IF xPoInicjalizacji THEN
		fnZapiszKomunikat(	sCalyKomunikat := '' ,
							sTypKomunikatu := 'E' ,
							sMnemonik := sMnemonik ,
							sMACAdres := sMACAdres ,
							sIDNadawcy := sIdInstancji ,
							sIDOdbiorcy := sIdAplikacji ,
							sDaneZapasowe := sDaneZapasowe ,
							sDane := fnKomunikatDaneError(xAktywny := FALSE , intKlasa := enumPPPSWezelClimatixPOL63xErrorKlasa.AlarmCzujnikaZewnetrznego , intNumer := enumPPPSWezelClimatixPOL63xError.AlarmCzujnikaZewnetrznego),
							arTablicaKomunikatow := arTablicaKomunikatow ,
							intTablicaKomunikatowZnacznikZapisu := intTablicaKomunikatowZnacznikZapisu ,
							intTablicaKomunikatowRozmiar := intTablicaKomunikatowRozmiar ,
							sWyslanyKomunikat := sWyslanyKomunikatDummy);
	END_IF
END_IF
// Alarm czujnika obwodu HC1
IF arErrorStan[enumPPPSWezelClimatixPOL63xError.AlarmCzujnikaZasilaniaObwoduHC1] <> enumAlarmWartosc.StanAlarmowy AND xBladBrakZmianyTemperaturyZewnetrznej AND arModbusStatusKomunikacji[bAdres] = enumModbusStatus.KomunikacjaPrawidlowa THEN
	arErrorStan[enumPPPSWezelClimatixPOL63xError.AlarmCzujnikaZasilaniaObwoduHC1] := enumAlarmWartosc.StanAlarmowy;
	arErrorKlasa[enumPPPSWezelClimatixPOL63xError.AlarmCzujnikaZasilaniaObwoduHC1] := enumPPPSWezelClimatixPOL63xErrorKlasa.AlarmCzujnikaZasilaniaObwoduHC1;
	IF xPoInicjalizacji THEN
		fnZapiszKomunikat(	sCalyKomunikat := '' ,
							sTypKomunikatu := 'E' ,
							sMnemonik := sMnemonik ,
							sMACAdres := sMACAdres ,
							sIDNadawcy := sIdInstancji ,
							sIDOdbiorcy := sIdAplikacji ,
							sDaneZapasowe := sDaneZapasowe ,
							sDane := fnKomunikatDaneError(xAktywny := TRUE , intKlasa := enumPPPSWezelClimatixPOL63xErrorKlasa.AlarmCzujnikaZasilaniaObwoduHC1 , intNumer := enumPPPSWezelClimatixPOL63xError.AlarmCzujnikaZasilaniaObwoduHC1),
							arTablicaKomunikatow := arTablicaKomunikatow ,
							intTablicaKomunikatowZnacznikZapisu := intTablicaKomunikatowZnacznikZapisu ,
							intTablicaKomunikatowRozmiar := intTablicaKomunikatowRozmiar ,
							sWyslanyKomunikat := sWyslanyKomunikatDummy);
	END_IF
END_IF
IF arErrorStan[enumPPPSWezelClimatixPOL63xError.AlarmCzujnikaZasilaniaObwoduHC1] <> enumAlarmWartosc.StanNormalny AND NOT xBladBrakZmianyTemperaturyZewnetrznej AND arModbusStatusKomunikacji[bAdres] = enumModbusStatus.KomunikacjaPrawidlowa THEN
	arErrorStan[enumPPPSWezelClimatixPOL63xError.AlarmCzujnikaZasilaniaObwoduHC1] := enumAlarmWartosc.StanNormalny;
	arErrorKlasa[enumPPPSWezelClimatixPOL63xError.AlarmCzujnikaZasilaniaObwoduHC1] := enumPPPSWezelClimatixPOL63xErrorKlasa.AlarmCzujnikaZasilaniaObwoduHC1;
	IF xPoInicjalizacji THEN
		fnZapiszKomunikat(	sCalyKomunikat := '' ,
							sTypKomunikatu := 'E' ,
							sMnemonik := sMnemonik ,
							sMACAdres := sMACAdres ,
							sIDNadawcy := sIdInstancji ,
							sIDOdbiorcy := sIdAplikacji ,
							sDaneZapasowe := sDaneZapasowe ,
							sDane := fnKomunikatDaneError(xAktywny := FALSE , intKlasa := enumPPPSWezelClimatixPOL63xErrorKlasa.AlarmCzujnikaZasilaniaObwoduHC1 , intNumer := enumPPPSWezelClimatixPOL63xError.AlarmCzujnikaZasilaniaObwoduHC1),
							arTablicaKomunikatow := arTablicaKomunikatow ,
							intTablicaKomunikatowZnacznikZapisu := intTablicaKomunikatowZnacznikZapisu ,
							intTablicaKomunikatowRozmiar := intTablicaKomunikatowRozmiar ,
							sWyslanyKomunikat := sWyslanyKomunikatDummy);
	END_IF
END_IF
// Alarm czujnika obwodu DHW
IF arErrorStan[enumPPPSWezelClimatixPOL63xError.AlarmCzujnikaZasilaniaObwoduDHW] <> enumAlarmWartosc.StanAlarmowy AND xBladBrakZmianyTemperaturyZewnetrznej AND arModbusStatusKomunikacji[bAdres] = enumModbusStatus.KomunikacjaPrawidlowa THEN
	arErrorStan[enumPPPSWezelClimatixPOL63xError.AlarmCzujnikaZasilaniaObwoduDHW] := enumAlarmWartosc.StanAlarmowy;
	arErrorKlasa[enumPPPSWezelClimatixPOL63xError.AlarmCzujnikaZasilaniaObwoduDHW] := enumPPPSWezelClimatixPOL63xErrorKlasa.AlarmCzujnikaZasilaniaObwoduDHW;
	IF xPoInicjalizacji THEN
		fnZapiszKomunikat(	sCalyKomunikat := '' ,
							sTypKomunikatu := 'E' ,
							sMnemonik := sMnemonik ,
							sMACAdres := sMACAdres ,
							sIDNadawcy := sIdInstancji ,
							sIDOdbiorcy := sIdAplikacji ,
							sDaneZapasowe := sDaneZapasowe ,
							sDane := fnKomunikatDaneError(xAktywny := TRUE , intKlasa := enumPPPSWezelClimatixPOL63xErrorKlasa.AlarmCzujnikaZasilaniaObwoduDHW , intNumer := enumPPPSWezelClimatixPOL63xError.AlarmCzujnikaZasilaniaObwoduDHW),
							arTablicaKomunikatow := arTablicaKomunikatow ,
							intTablicaKomunikatowZnacznikZapisu := intTablicaKomunikatowZnacznikZapisu ,
							intTablicaKomunikatowRozmiar := intTablicaKomunikatowRozmiar ,
							sWyslanyKomunikat := sWyslanyKomunikatDummy);
	END_IF
END_IF
IF arErrorStan[enumPPPSWezelClimatixPOL63xError.AlarmCzujnikaZasilaniaObwoduDHW] <> enumAlarmWartosc.StanNormalny AND NOT xBladBrakZmianyTemperaturyZewnetrznej AND arModbusStatusKomunikacji[bAdres] = enumModbusStatus.KomunikacjaPrawidlowa THEN
	arErrorStan[enumPPPSWezelClimatixPOL63xError.AlarmCzujnikaZasilaniaObwoduDHW] := enumAlarmWartosc.StanNormalny;
	arErrorKlasa[enumPPPSWezelClimatixPOL63xError.AlarmCzujnikaZasilaniaObwoduDHW] := enumPPPSWezelClimatixPOL63xErrorKlasa.AlarmCzujnikaZasilaniaObwoduDHW;
	IF xPoInicjalizacji THEN
		fnZapiszKomunikat(	sCalyKomunikat := '' ,
							sTypKomunikatu := 'E' ,
							sMnemonik := sMnemonik ,
							sMACAdres := sMACAdres ,
							sIDNadawcy := sIdInstancji ,
							sIDOdbiorcy := sIdAplikacji ,
							sDaneZapasowe := sDaneZapasowe ,
							sDane := fnKomunikatDaneError(xAktywny := FALSE , intKlasa := enumPPPSWezelClimatixPOL63xErrorKlasa.AlarmCzujnikaZasilaniaObwoduDHW , intNumer := enumPPPSWezelClimatixPOL63xError.AlarmCzujnikaZasilaniaObwoduDHW),
							arTablicaKomunikatow := arTablicaKomunikatow ,
							intTablicaKomunikatowZnacznikZapisu := intTablicaKomunikatowZnacznikZapisu ,
							intTablicaKomunikatowRozmiar := intTablicaKomunikatowRozmiar ,
							sWyslanyKomunikat := sWyslanyKomunikatDummy);
	END_IF
END_IF
// Alarm braku osiągnięcia zadanej temperatury zasilania obwodu HC1
IF arErrorStan[enumPPPSWezelClimatixPOL63xError.AlarmBrakuOsiagnieciaTemperaturyHC1] <> enumAlarmWartosc.StanAlarmowy AND xBladBrakZmianyTemperaturyZewnetrznej AND arModbusStatusKomunikacji[bAdres] = enumModbusStatus.KomunikacjaPrawidlowa THEN
	arErrorStan[enumPPPSWezelClimatixPOL63xError.AlarmBrakuOsiagnieciaTemperaturyHC1] := enumAlarmWartosc.StanAlarmowy;
	arErrorKlasa[enumPPPSWezelClimatixPOL63xError.AlarmBrakuOsiagnieciaTemperaturyHC1] := enumPPPSWezelClimatixPOL63xErrorKlasa.AlarmBrakuOsiagnieciaTemperaturyHC1;
	IF xPoInicjalizacji THEN
		fnZapiszKomunikat(	sCalyKomunikat := '' ,
							sTypKomunikatu := 'E' ,
							sMnemonik := sMnemonik ,
							sMACAdres := sMACAdres ,
							sIDNadawcy := sIdInstancji ,
							sIDOdbiorcy := sIdAplikacji ,
							sDaneZapasowe := sDaneZapasowe ,
							sDane := fnKomunikatDaneError(xAktywny := TRUE , intKlasa := enumPPPSWezelClimatixPOL63xErrorKlasa.AlarmBrakuOsiagnieciaTemperaturyHC1 , intNumer := enumPPPSWezelClimatixPOL63xError.AlarmBrakuOsiagnieciaTemperaturyHC1),
							arTablicaKomunikatow := arTablicaKomunikatow ,
							intTablicaKomunikatowZnacznikZapisu := intTablicaKomunikatowZnacznikZapisu ,
							intTablicaKomunikatowRozmiar := intTablicaKomunikatowRozmiar ,
							sWyslanyKomunikat := sWyslanyKomunikatDummy);
	END_IF
END_IF
IF arErrorStan[enumPPPSWezelClimatixPOL63xError.AlarmBrakuOsiagnieciaTemperaturyHC1] <> enumAlarmWartosc.StanNormalny AND NOT xBladBrakZmianyTemperaturyZewnetrznej AND arModbusStatusKomunikacji[bAdres] = enumModbusStatus.KomunikacjaPrawidlowa THEN
	arErrorStan[enumPPPSWezelClimatixPOL63xError.AlarmBrakuOsiagnieciaTemperaturyHC1] := enumAlarmWartosc.StanNormalny;
	arErrorKlasa[enumPPPSWezelClimatixPOL63xError.AlarmBrakuOsiagnieciaTemperaturyHC1] := enumPPPSWezelClimatixPOL63xErrorKlasa.AlarmBrakuOsiagnieciaTemperaturyHC1;
	IF xPoInicjalizacji THEN
		fnZapiszKomunikat(	sCalyKomunikat := '' ,
							sTypKomunikatu := 'E' ,
							sMnemonik := sMnemonik ,
							sMACAdres := sMACAdres ,
							sIDNadawcy := sIdInstancji ,
							sIDOdbiorcy := sIdAplikacji ,
							sDaneZapasowe := sDaneZapasowe ,
							sDane := fnKomunikatDaneError(xAktywny := FALSE , intKlasa := enumPPPSWezelClimatixPOL63xErrorKlasa.AlarmBrakuOsiagnieciaTemperaturyHC1 , intNumer := enumPPPSWezelClimatixPOL63xError.AlarmBrakuOsiagnieciaTemperaturyHC1),
							arTablicaKomunikatow := arTablicaKomunikatow ,
							intTablicaKomunikatowZnacznikZapisu := intTablicaKomunikatowZnacznikZapisu ,
							intTablicaKomunikatowRozmiar := intTablicaKomunikatowRozmiar ,
							sWyslanyKomunikat := sWyslanyKomunikatDummy);
	END_IF
END_IF
// Alarm braku osiągnięcia zadanej temperatury zasilania obwodu DHW
IF arErrorStan[enumPPPSWezelClimatixPOL63xError.AlarmBrakuOsiagnieciaTemperaturyDHW] <> enumAlarmWartosc.StanAlarmowy AND xBladBrakZmianyTemperaturyZewnetrznej AND arModbusStatusKomunikacji[bAdres] = enumModbusStatus.KomunikacjaPrawidlowa THEN
	arErrorStan[enumPPPSWezelClimatixPOL63xError.AlarmBrakuOsiagnieciaTemperaturyDHW] := enumAlarmWartosc.StanAlarmowy;
	arErrorKlasa[enumPPPSWezelClimatixPOL63xError.AlarmBrakuOsiagnieciaTemperaturyDHW] := enumPPPSWezelClimatixPOL63xErrorKlasa.AlarmBrakuOsiagnieciaTemperaturyDHW;
	IF xPoInicjalizacji THEN
		fnZapiszKomunikat(	sCalyKomunikat := '' ,
							sTypKomunikatu := 'E' ,
							sMnemonik := sMnemonik ,
							sMACAdres := sMACAdres ,
							sIDNadawcy := sIdInstancji ,
							sIDOdbiorcy := sIdAplikacji ,
							sDaneZapasowe := sDaneZapasowe ,
							sDane := fnKomunikatDaneError(xAktywny := TRUE , intKlasa := enumPPPSWezelClimatixPOL63xErrorKlasa.AlarmBrakuOsiagnieciaTemperaturyDHW , intNumer := enumPPPSWezelClimatixPOL63xError.AlarmBrakuOsiagnieciaTemperaturyDHW),
							arTablicaKomunikatow := arTablicaKomunikatow ,
							intTablicaKomunikatowZnacznikZapisu := intTablicaKomunikatowZnacznikZapisu ,
							intTablicaKomunikatowRozmiar := intTablicaKomunikatowRozmiar ,
							sWyslanyKomunikat := sWyslanyKomunikatDummy);
	END_IF
END_IF
IF arErrorStan[enumPPPSWezelClimatixPOL63xError.AlarmBrakuOsiagnieciaTemperaturyDHW] <> enumAlarmWartosc.StanNormalny AND NOT xBladBrakZmianyTemperaturyZewnetrznej AND arModbusStatusKomunikacji[bAdres] = enumModbusStatus.KomunikacjaPrawidlowa THEN
	arErrorStan[enumPPPSWezelClimatixPOL63xError.AlarmBrakuOsiagnieciaTemperaturyDHW] := enumAlarmWartosc.StanNormalny;
	arErrorKlasa[enumPPPSWezelClimatixPOL63xError.AlarmBrakuOsiagnieciaTemperaturyDHW] := enumPPPSWezelClimatixPOL63xErrorKlasa.AlarmBrakuOsiagnieciaTemperaturyDHW;
	IF xPoInicjalizacji THEN
		fnZapiszKomunikat(	sCalyKomunikat := '' ,
							sTypKomunikatu := 'E' ,
							sMnemonik := sMnemonik ,
							sMACAdres := sMACAdres ,
							sIDNadawcy := sIdInstancji ,
							sIDOdbiorcy := sIdAplikacji ,
							sDaneZapasowe := sDaneZapasowe ,
							sDane := fnKomunikatDaneError(xAktywny := FALSE , intKlasa := enumPPPSWezelClimatixPOL63xErrorKlasa.AlarmBrakuOsiagnieciaTemperaturyDHW , intNumer := enumPPPSWezelClimatixPOL63xError.AlarmBrakuOsiagnieciaTemperaturyDHW),
							arTablicaKomunikatow := arTablicaKomunikatow ,
							intTablicaKomunikatowZnacznikZapisu := intTablicaKomunikatowZnacznikZapisu ,
							intTablicaKomunikatowRozmiar := intTablicaKomunikatowRozmiar ,
							sWyslanyKomunikat := sWyslanyKomunikatDummy);
	END_IF
END_IF
// Alarm braku wymaganej ilości pomiarów do obliczenia średniej temperatury
IF arErrorStan[enumPPPSWezelClimatixPOL63xError.BladIloscPomiarowTemperatury] <> enumAlarmWartosc.StanAlarmowy AND xBladIloscPomiarowTemperatury THEN
	arErrorStan[enumPPPSWezelClimatixPOL63xError.BladIloscPomiarowTemperatury] := enumAlarmWartosc.StanAlarmowy;
	arErrorKlasa[enumPPPSWezelClimatixPOL63xError.BladIloscPomiarowTemperatury] := enumPPPSWezelClimatixPOL63xError.BladIloscPomiarowTemperatury;
	IF xPoInicjalizacji THEN
		fnZapiszKomunikat(	sCalyKomunikat := '' ,
							sTypKomunikatu := 'E' ,
							sMnemonik := sMnemonik ,
							sMACAdres := sMACAdres ,
							sIDNadawcy := sIdInstancji ,
							sIDOdbiorcy := sIdAplikacji ,
							sDaneZapasowe := sDaneZapasowe ,
							sDane := fnKomunikatDaneError(xAktywny := TRUE , intKlasa := enumPPPSWezelClimatixPOL63xError.BladIloscPomiarowTemperatury , intNumer := enumPPPSWezelClimatixPOL63xError.BladIloscPomiarowTemperatury),
							arTablicaKomunikatow := arTablicaKomunikatow ,
							intTablicaKomunikatowZnacznikZapisu := intTablicaKomunikatowZnacznikZapisu ,
							intTablicaKomunikatowRozmiar := intTablicaKomunikatowRozmiar ,
							sWyslanyKomunikat := sWyslanyKomunikatDummy);
	END_IF
END_IF

// Sprawdzanie czy pomiar temperatury zewnętrznej działa (alarm jest generowany, jeśli odczyt nie zmienił wartości w przeciągu 12h)
IF xInstalacjaHC1 THEN
	IF rTemperaturaZewnetrznaPamiec = rTemperaturaZewnetrzna THEN
		xBrakZmianyTemperaturyZewnetrznej := TRUE;
	ELSE
		xBrakZmianyTemperaturyZewnetrznej := FALSE;	
	END_IF
	fbBrakZmianyTemperaturyZewnetrznejTimer(IN := xBrakZmianyTemperaturyZewnetrznej, PT := T#12H);
	rTemperaturaZewnetrznaPamiec := rTemperaturaZewnetrzna;
	IF fbBrakZmianyTemperaturyZewnetrznejTimer.Q THEN
		xBladBrakZmianyTemperaturyZewnetrznej := TRUE;
	ELSE
		xBladBrakZmianyTemperaturyZewnetrznej := FALSE;
	END_IF
END_IF

// Sprawdzanie czy pomiar temperatury zasilania obwodu HC1 działa (alarm jest generowany, jeśli odczyt nie zmienił wartości w przeciągu 12h)
IF xInstalacjaHC1 THEN
	IF rTemperaturaZasilaniaObwoduHC1Pamiec = rTemperaturaZasilaniaObwoduHC1 THEN
		xBrakZmianyTemperaturyZasilaniaObwoduHC1 := TRUE;
	ELSE
		xBrakZmianyTemperaturyZasilaniaObwoduHC1 := FALSE;	
	END_IF
	fbBrakZmianyTemperaturyZasilaniaObwoduHC1Timer(IN := xBrakZmianyTemperaturyZasilaniaObwoduHC1, PT := T#12H);
	rTemperaturaZasilaniaObwoduHC1Pamiec := rTemperaturaZasilaniaObwoduHC1;
	IF fbBrakZmianyTemperaturyZasilaniaObwoduHC1Timer.Q THEN
		xBladBrakZmianyTemperaturyZasilaniaObwoduHC1 := TRUE;
	ELSE
		xBladBrakZmianyTemperaturyZasilaniaObwoduHC1 := FALSE;
	END_IF
END_IF

// Sprawdzanie czy pomiar temperatury zasilania obwodu DHW działa (alarm jest generowany, jeśli odczyt nie zmienił wartości w przeciągu 12h)
IF xInstalacjaDHW THEN
	IF rTemperaturaZasilaniaObwoduDHWPamiec = rTemperaturaZasilaniaBudynekDHW THEN
		xBrakZmianyTemperaturyZasilaniaObwoduDHW := TRUE;
	ELSE
		xBrakZmianyTemperaturyZasilaniaObwoduDHW := FALSE;	
	END_IF
	fbBrakZmianyTemperaturyZasilaniaObwoduDHWTimer(IN := xBrakZmianyTemperaturyZasilaniaObwoduDHW, PT := T#12H);
	rTemperaturaZasilaniaObwoduDHWPamiec := rTemperaturaZasilaniaBudynekDHW;
	IF fbBrakZmianyTemperaturyZasilaniaObwoduDHWTimer.Q THEN
		xBladBrakZmianyTemperaturyZasilaniaObwoduDHW := TRUE;
	ELSE
		xBladBrakZmianyTemperaturyZasilaniaObwoduDHW := FALSE;
	END_IF
END_IF

// Sprawdzanie czy została osiągnęta zadana temperatura zasilania obwodu HC1
IF xInstalacjaHC1 THEN
	IF rTemperaturaZasilaniaObwoduHC1 < rTemperaturaGrzaniaNastawionaHC1 THEN
		xBrakOsiagnieciaTemperauryZadanejHC1 := TRUE;
	ELSE
		xBrakOsiagnieciaTemperauryZadanejHC1 := FALSE;	
	END_IF
	fbBrakOsiagnieciaTemperauryZadanejHC1Timer(IN := xBrakOsiagnieciaTemperauryZadanejHC1, PT := T#3H);
	IF fbBrakOsiagnieciaTemperauryZadanejHC1Timer.Q THEN
		xBladBrakOsiagnieciaTemperauryZadanejHC1 := TRUE;
	ELSE
		xBladBrakOsiagnieciaTemperauryZadanejHC1 := FALSE;
	END_IF
END_IF

// Sprawdzanie czy została osiągnęta zadana temperatura zasilania obwodu DHW
IF xInstalacjaDHW THEN
	IF rTemperaturaZasilaniaBudynekDHW < rTemperaturaGrzaniaNastawionaDHW THEN
		xBrakOsiagnieciaTemperauryZadanejDHW := TRUE;
	ELSE
		xBrakOsiagnieciaTemperauryZadanejDHW := FALSE;	
	END_IF
	fbBrakOsiagnieciaTemperauryZadanejDHWTimer(IN := xBrakOsiagnieciaTemperauryZadanejDHW, PT := T#3H);
	IF fbBrakOsiagnieciaTemperauryZadanejDHWTimer.Q THEN
		xBladBrakOsiagnieciaTemperauryZadanejDHW := TRUE;
	ELSE
		xBladBrakOsiagnieciaTemperauryZadanejDHW := FALSE;
	END_IF
END_IF
          
END_FUNCTION_BLOCK
